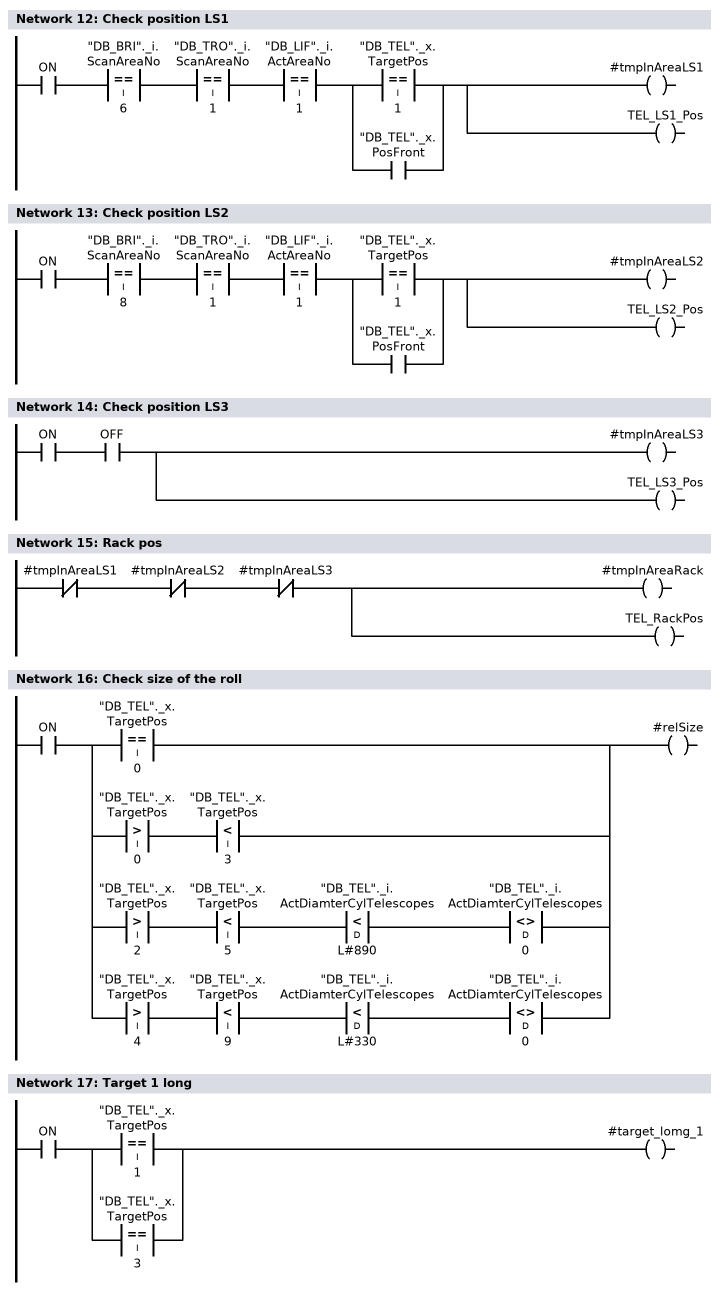
[picture p309: Axis_TEL_Control networks 12-17]
NETWORK
TITLE = Check position LS1
      A     "ON";
      A(;
      L     "DB_BRI"._i.ScanAreaNo;
      L     6;
      ==I;
      );
      A(;
      L     "DB_TRO"._i.ScanAreaNo;
      L     1;
      ==I;
      );
      A(;
      L     "DB_LIF"._i.ActAreaNo;
      L     1;
      ==I;
      );
      A(;
      O(;
      L     "DB_TEL"._x.TargetPos;
      L     1;
      ==I;
      );
      O     "DB_TEL"._x.PosFront;
      );
      =     #tmpInAreaLS1;
      =     "TEL_LS1_Pos";
NETWORK
TITLE = Check position LS2
      A     "ON";
      A(;
      L     "DB_BRI"._i.ScanAreaNo;
      L     8;
      ==I;
      );
      A(;
      L     "DB_TRO"._i.ScanAreaNo;
      L     1;
      ==I;
      );
      A(;
      L     "DB_LIF"._i.ActAreaNo;
      L     1;
      ==I;
      );
      A(;
      O(;
      L     "DB_TEL"._x.TargetPos;
      L     1;
      ==I;
      );
      O     "DB_TEL"._x.PosFront;
      );
      =     #tmpInAreaLS2;
      =     "TEL_LS2_Pos";
NETWORK
TITLE = Check position LS3
      A     "ON";
      A     "OFF";
      =     #tmpInAreaLS3;
      =     "TEL_LS3_Pos";
NETWORK
TITLE = Rack pos
      AN    #tmpInAreaLS1;
      AN    #tmpInAreaLS2;
      AN    #tmpInAreaLS3;
      =     #tmpInAreaRack;
      =     "TEL_RackPos";
NETWORK
TITLE = Check size of the roll
      A     "ON";
      A(;
      O(;
      L     "DB_TEL"._x.TargetPos;
      L     0;
      ==I;
      );
      O;
      A(;
      L     "DB_TEL"._x.TargetPos;
      L     0;
      >I;
      );
      A(;
      L     "DB_TEL"._x.TargetPos;
      L     3;
      <I;
      );
      O;
      A(;
      L     "DB_TEL"._x.TargetPos;
      L     2;
      >I;
      );
      A(;
      L     "DB_TEL"._x.TargetPos;
      L     5;
      <I;
      );
      A(;
      L     "DB_TEL"._i.ActDiamterCylTelescopes;
      L     L#890;
      <D;
      );
      A(;
      L     "DB_TEL"._i.ActDiamterCylTelescopes;
      L     0;
      <>D;
      );
      O;
      A(;
      L     "DB_TEL"._x.TargetPos;
      L     4;
      >I;
      );
      A(;
      L     "DB_TEL"._x.TargetPos;
      L     9;
      <I;
      );
      A(;
      L     "DB_TEL"._i.ActDiamterCylTelescopes;
      L     L#330;
      <D;
      );
      A(;
      L     "DB_TEL"._i.ActDiamterCylTelescopes;
      L     0;
      <>D;
      );
      );
      =     #relSize;
NETWORK
TITLE = Target 1 long
      A     "ON";
      A(;
      O(;
      L     "DB_TEL"._x.TargetPos;
      L     1;
      ==I;
      );
      O(;
      L     "DB_TEL"._x.TargetPos;
      L     3;
      ==I;
      );
      );
      =     #target_lomg_1;
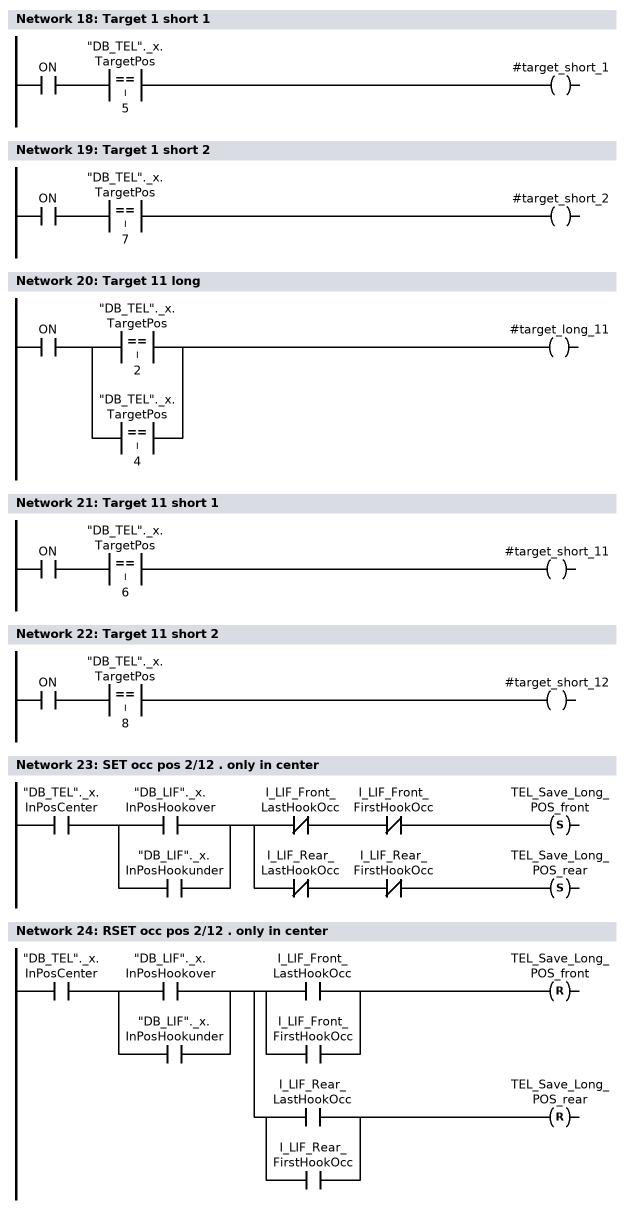
NETWORK
TITLE = Target 1 short 1
      A     "ON";
      A(;
      L     "DB_TEL"._x.TargetPos;
      L     5;
      ==I;
      );
      =     #target_short_1;
NETWORK
TITLE = Target 1 short 2
      A     "ON";
      A(;
      L     "DB_TEL"._x.TargetPos;
      L     7;
      ==I;
      );
      =     #target_short_2;
NETWORK
TITLE = Target 11 long
      A     "ON";
      A(;
      O(;
      L     "DB_TEL"._x.TargetPos;
      L     2;
      ==I;
      );
      O(;
      L     "DB_TEL"._x.TargetPos;
      L     4;
      ==I;
      );
      );
      =     #target_long_11;
NETWORK
TITLE = Target 11 short 1
      A     "ON";
      A(;
      L     "DB_TEL"._x.TargetPos;
      L     6;
      ==I;
      );
      =     #target_short_11;
NETWORK
TITLE = Target 11 short 2
      A     "ON";
      A(;
      L     "DB_TEL"._x.TargetPos;
      L     8;
      ==I;
      );
      =     #target_short_12;
NETWORK
TITLE = SET occ pos 2/12 . only in center
      A     "DB_TEL"._x.InPosCenter;
      A(;
      O     "DB_LIF"._x.InPosHookover;
      O     "DB_LIF"._x.InPosHookunder;
      );
      =     L 20.0;
      A     L 20.0;
      AN    "I_LIF_Front_LastHookOcc";
      AN    "I_LIF_Front_FirstHookOcc";
      S     "TEL_Save_Long_POS_front";
      A     L 20.0;
      AN    "I_LIF_Rear_LastHookOcc";
      AN    "I_LIF_Rear_FirstHookOcc";
      S     "TEL_Save_Long_POS_rear";
NETWORK
TITLE = RSET occ pos 2/12 . only in center
      A     "DB_TEL"._x.InPosCenter;
      A(;
      O     "DB_LIF"._x.InPosHookover;
      O     "DB_LIF"._x.InPosHookunder;
      );
      =     L 20.0;
      A     L 20.0;
      A(;
      O     "I_LIF_Front_LastHookOcc";
      O     "I_LIF_Front_FirstHookOcc";
      );
      R     "TEL_Save_Long_POS_front";
      A     L 20.0;
      A(;
      O     "I_LIF_Rear_LastHookOcc";
      O     "I_LIF_Rear_FirstHookOcc";
      );
      R     "TEL_Save_Long_POS_rear";
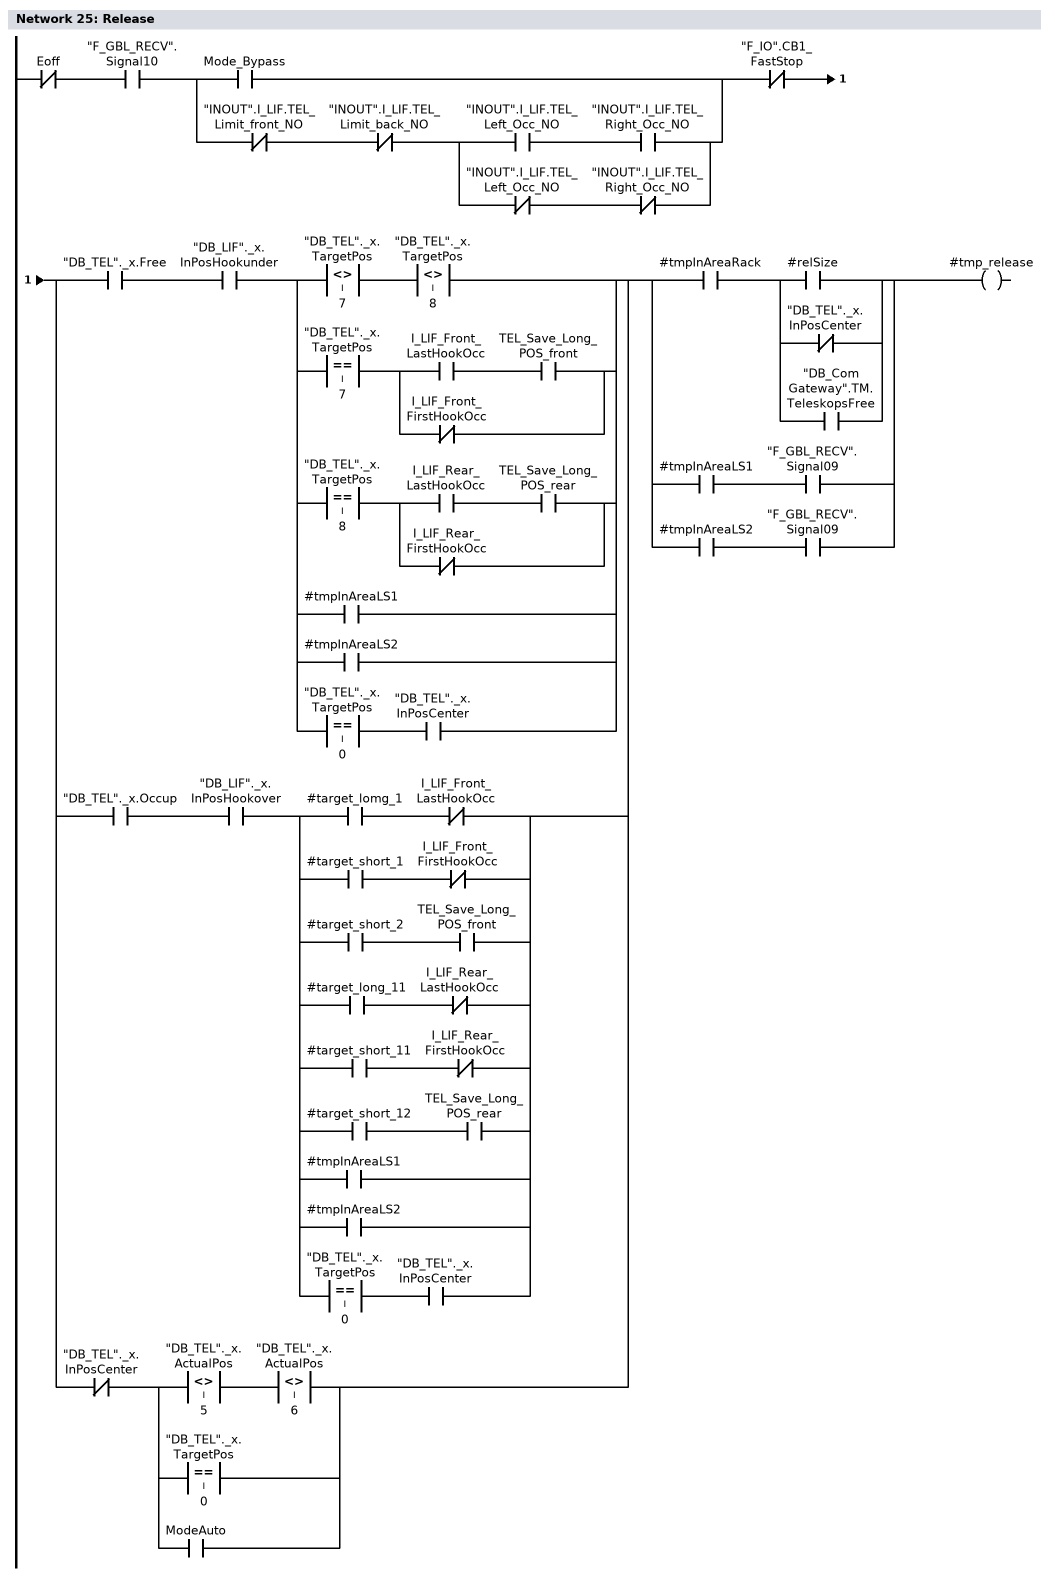
NETWORK
TITLE = Release
//DB400.DBX43.0 LIFT Wago
      AN    "Eoff";
      A     "F_GBL_RECV".Signal10;
      A(;
      O     "Mode_Bypass";
      O;
      AN    "INOUT".I_LIF.TEL_Limit_front_NO;
      AN    "INOUT".I_LIF.TEL_Limit_back_NO;
      A(;
      A     "INOUT".I_LIF.TEL_Left_Occ_NO;
      A     "INOUT".I_LIF.TEL_Right_Occ_NO;
      O;
      AN    "INOUT".I_LIF.TEL_Left_Occ_NO;
      AN    "INOUT".I_LIF.TEL_Right_Occ_NO;
      );
      );
      AN    "F_IO".CB1_FastStop;
      A(;
      A     "DB_TEL"._x.Free;
      A     "DB_LIF"._x.InPosHookunder;
      A(;
      A(;
      L     "DB_TEL"._x.TargetPos;
      L     7;
      <>I;
      );
      A(;
      L     "DB_TEL"._x.TargetPos;
      L     8;
      <>I;
      );
      O;
      A(;
      L     "DB_TEL"._x.TargetPos;
      L     7;
      ==I;
      );
      A(;
      A     "I_LIF_Front_LastHookOcc";
      A     "TEL_Save_Long_POS_front";
      ON    "I_LIF_Front_FirstHookOcc";
      );
      O;
      A(;
      L     "DB_TEL"._x.TargetPos;
      L     8;
      ==I;
      );
      A(;
      A     "I_LIF_Rear_LastHookOcc";
      A     "TEL_Save_Long_POS_rear";
      ON    "I_LIF_Rear_FirstHookOcc";
      );
      O     #tmpInAreaLS1;
      O     #tmpInAreaLS2;
      O;
      A(;
      L     "DB_TEL"._x.TargetPos;
      L     0;
      ==I;
      );
      A     "DB_TEL"._x.InPosCenter;
      );
      O;
      A     "DB_TEL"._x.Occup;
      A     "DB_LIF"._x.InPosHookover;
      A(;
      A     #target_lomg_1;
      AN    "I_LIF_Front_LastHookOcc";
      O;
      A     #target_short_1;
      AN    "I_LIF_Front_FirstHookOcc";
      O;
      A     #target_short_2;
      A     "TEL_Save_Long_POS_front";
      O;
      A     #target_long_11;
      AN    "I_LIF_Rear_LastHookOcc";
      O;
      A     #target_short_11;
      AN    "I_LIF_Rear_FirstHookOcc";
      O;
      A     #target_short_12;
      A     "TEL_Save_Long_POS_rear";
      O     #tmpInAreaLS1;
      O     #tmpInAreaLS2;
      O;
      A(;
      L     "DB_TEL"._x.TargetPos;
      L     0;
      ==I;
      );
      A     "DB_TEL"._x.InPosCenter;
      );
      O;
      AN    "DB_TEL"._x.InPosCenter;
      A(;
      A(;
      L     "DB_TEL"._x.ActualPos;
      L     5;
      <>I;
      );
      A(;
      L     "DB_TEL"._x.ActualPos;
      L     6;
      <>I;
      );
      O(;
      L     "DB_TEL"._x.TargetPos;
      L     0;
      ==I;
      );
      O     "ModeAuto";
      );
      );
      A(;
      A     #tmpInAreaRack;
      A(;
      O     #relSize;
      ON    "DB_TEL"._x.InPosCenter;
      O     "DB_ComGateway".TM.TeleskopsFree;
      );
      O;
      A     #tmpInAreaLS1;
      A     "F_GBL_RECV".Signal09;
      O;
      A     #tmpInAreaLS2;
      A     "F_GBL_RECV".Signal09;
      );
      =     #tmp_release;
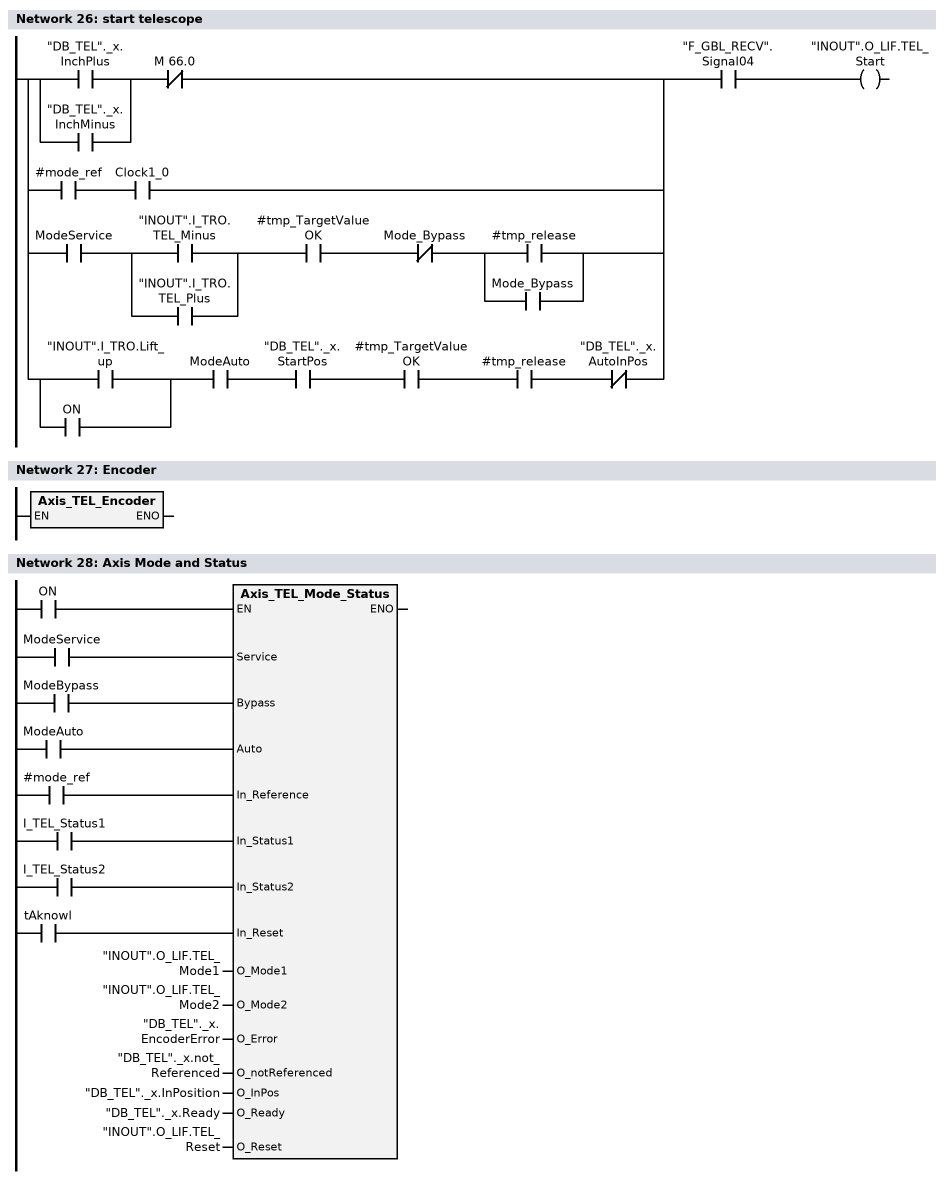
NETWORK
TITLE = start telescope 
      A(;
      A(;
      O     "DB_TEL"._x.InchPlus;
      O     "DB_TEL"._x.InchMinus;
      );
      AN    M 66.0;
      O;
      A     #mode_ref;
      A     "Clock1_0";
      O;
      A     "ModeService";
      A(;
      O     "INOUT".I_TRO.TEL_Minus;
      O     "INOUT".I_TRO.TEL_Plus;
      );
      A     #tmp_TargetValueOK;
      AN    "Mode_Bypass";
      A(;
      O     #tmp_release;
      O     "Mode_Bypass";
      );
      O;
      A(;
      O     "INOUT".I_TRO.Lift_up;
      O     "ON";
      );
      A     "ModeAuto";
      A     "DB_TEL"._x.StartPos;
      A     #tmp_TargetValueOK;
      A     #tmp_release;
      AN    "DB_TEL"._x.AutoInPos;
      );
      A     "F_GBL_RECV".Signal04;
      =     "INOUT".O_LIF.TEL_Start;
NETWORK
TITLE = Encoder
      CALL  "Axis_TEL_Encoder";
      NOP   0;
NETWORK
TITLE = Axis Mode and Status
      A     "ModeService";
      =     L 20.0;
      BLD   103;
      A     "ModeBypass";
      =     L 20.1;
      BLD   103;
      A     "ModeAuto";
      =     L 20.2;
      BLD   103;
      A     #mode_ref;
      =     L 20.3;
      BLD   103;
      A     "I_TEL_Status1";
      =     L 20.4;
      BLD   103;
      A     "I_TEL_Status2";
      =     L 20.5;
      BLD   103;
      A     "tAknowl";
      =     L 20.6;
      BLD   103;
      A     "ON";
      JNB   _00b;
      CALL  "Axis_TEL_Mode_Status" (
           Service                  := L 20.0,
           Bypass                   := L 20.1,
           Auto                     := L 20.2,
           In_Reference             := L 20.3,
           In_Status1               := L 20.4,
           In_Status2               := L 20.5,
           In_Reset                 := L 20.6,
           O_Mode1                  := "INOUT".O_LIF.TEL_Mode1,
           O_Mode2                  := "INOUT".O_LIF.TEL_Mode2,
           O_Error                  := "DB_TEL"._x.EncoderError,
           O_notReferenced          := "DB_TEL"._x.not_Referenced,
           O_InPos                  := "DB_TEL"._x.InPosition,
           O_Ready                  := "DB_TEL"._x.Ready,
           O_Reset                  := "INOUT".O_LIF.TEL_Reset);
_00b: NOP   0;
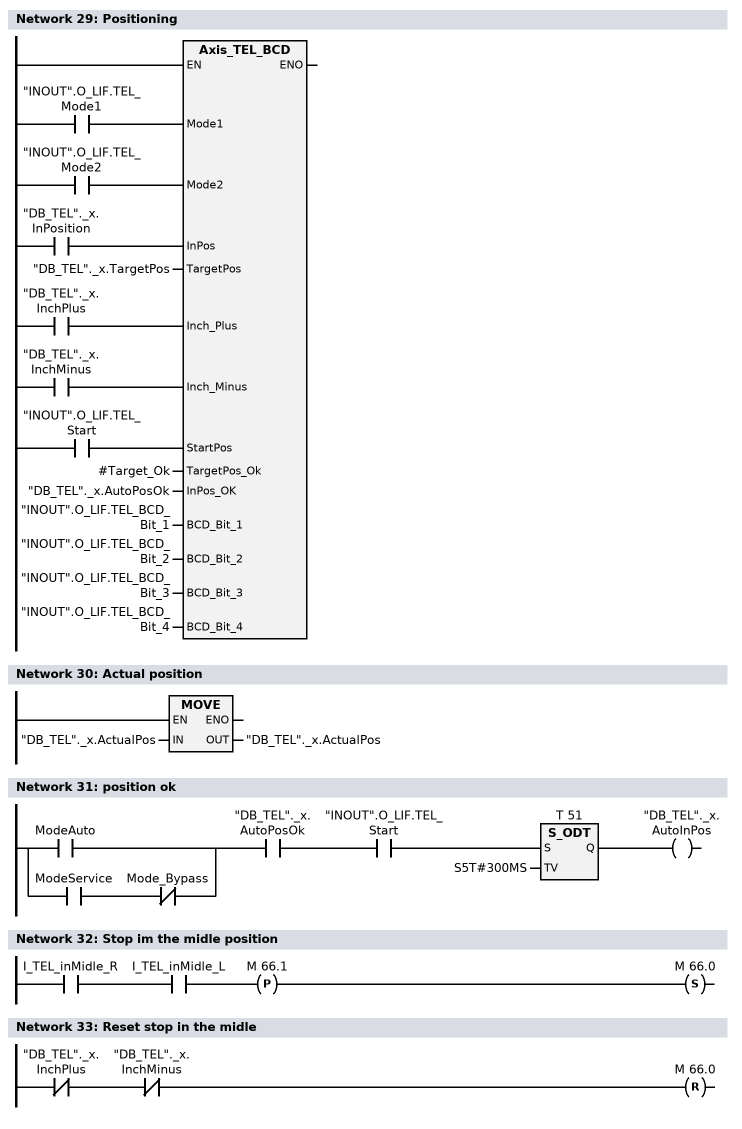
NETWORK
TITLE = Positioning
      A     "INOUT".O_LIF.TEL_Mode1;
      =     L 20.0;
      BLD   103;
      A     "INOUT".O_LIF.TEL_Mode2;
      =     L 20.1;
      BLD   103;
      A     "DB_TEL"._x.InPosition;
      =     L 20.2;
      BLD   103;
      A     "DB_TEL"._x.InchPlus;
      =     L 20.3;
      BLD   103;
      A     "DB_TEL"._x.InchMinus;
      =     L 20.4;
      BLD   103;
      A     "INOUT".O_LIF.TEL_Start;
      =     L 20.5;
      BLD   103;
      CALL  "Axis_TEL_BCD" (
           Mode1                    := L 20.0,
           Mode2                    := L 20.1,
           InPos                    := L 20.2,
           TargetPos                := "DB_TEL"._x.TargetPos,
           Inch_Plus                := L 20.3,
           Inch_Minus               := L 20.4,
           StartPos                 := L 20.5,
           TargetPos_Ok             := #Target_Ok,
           InPos_OK                 := "DB_TEL"._x.AutoPosOk,
           BCD_Bit_1                := "INOUT".O_LIF.TEL_BCD_Bit_1,
           BCD_Bit_2                := "INOUT".O_LIF.TEL_BCD_Bit_2,
           BCD_Bit_3                := "INOUT".O_LIF.TEL_BCD_Bit_3,
           BCD_Bit_4                := "INOUT".O_LIF.TEL_BCD_Bit_4);
      NOP   0;
NETWORK
TITLE = Actual position
      L     "DB_TEL"._x.ActualPos;
      T     "DB_TEL"._x.ActualPos;
      NOP   0;
NETWORK
TITLE = position ok
      A(;
      O     "ModeAuto";
      O;
      A     "ModeService";
      AN    "Mode_Bypass";
      );
      A     "DB_TEL"._x.AutoPosOk;
      A     "INOUT".O_LIF.TEL_Start;
      L     S5T#300MS;
      SD    T 51;
      NOP   0;
      NOP   0;
      NOP   0;
      A     T 51;
      =     "DB_TEL"._x.AutoInPos;
NETWORK
TITLE = Stop im the midle position
      A     "I_TEL_inMidle_R";
      A     "I_TEL_inMidle_L";
      FP    M 66.1;
      S     M 66.0;
NETWORK
TITLE = Reset stop in the midle
      AN    "DB_TEL"._x.InchPlus;
      AN    "DB_TEL"._x.InchMinus;
      R     M 66.0;
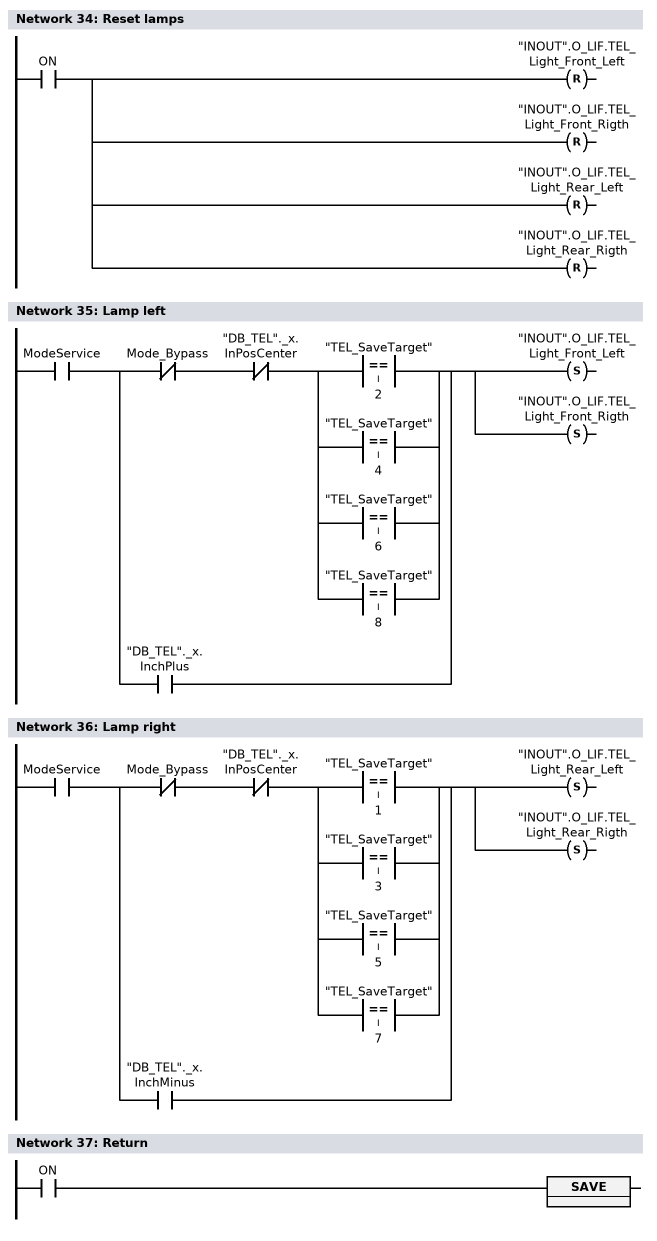
NETWORK
TITLE = Reset lamps
      A     "ON";
      R     "INOUT".O_LIF.TEL_Light_Front_Left;
      R     "INOUT".O_LIF.TEL_Light_Front_Rigth;
      R     "INOUT".O_LIF.TEL_Light_Rear_Left;
      R     "INOUT".O_LIF.TEL_Light_Rear_Rigth;
NETWORK
TITLE = Lamp left
      A     "ModeService";
      A(;
      AN    "Mode_Bypass";
      AN    "DB_TEL"._x.InPosCenter;
      A(;
      O(;
      L     "TEL_SaveTarget";
      L     2;
      ==I;
      );
      O(;
      L     "TEL_SaveTarget";
      L     4;
      ==I;
      );
      O(;
      L     "TEL_SaveTarget";
      L     6;
      ==I;
      );
      O(;
      L     "TEL_SaveTarget";
      L     8;
      ==I;
      );
      );
      O     "DB_TEL"._x.InchPlus;
      );
      S     "INOUT".O_LIF.TEL_Light_Front_Left;
      S     "INOUT".O_LIF.TEL_Light_Front_Rigth;
NETWORK
TITLE = Lamp right
      A     "ModeService";
      A(;
      AN    "Mode_Bypass";
      AN    "DB_TEL"._x.InPosCenter;
      A(;
      O(;
      L     "TEL_SaveTarget";
      L     1;
      ==I;
      );
      O(;
      L     "TEL_SaveTarget";
      L     3;
      ==I;
      );
      O(;
      L     "TEL_SaveTarget";
      L     5;
      ==I;
      );
      O(;
      L     "TEL_SaveTarget";
      L     7;
      ==I;
      );
      );
      O     "DB_TEL"._x.InchMinus;
      );
      S     "INOUT".O_LIF.TEL_Light_Rear_Left;
      S     "INOUT".O_LIF.TEL_Light_Rear_Rigth;
NETWORK
TITLE = Return
      A     "ON";
      SAVE;
END_FUNCTION

FUNCTION "Axis_TEL_Speed" : VOID	// FC 233
VERSION : 0.1
BEGIN
NETWORK
TITLE =
END_FUNCTION

FUNCTION "Axis_TEL_Scan" : VOID	// FC 234
TITLE = Axis TELESCOPES Scan
VERSION : 0.1
VAR_TEMP
  tmp_di_StopWindow : DINT ;
  tmp_di_PosWindow : DINT ;
  tmp_win : DINT ;
  tmp_AreaNo : INT ;
  tmp_InPos : BOOL ;
  tmp_InArea : BOOL ;
  tmp_x_InStopPosMan : BOOL ;
  tmp_x_InStopPosAuto : BOOL ;
  tmp_x_InStopCenterPos : BOOL ;
  tmp_OccFsPos1 : BOOL ;
  tmp_OccBsPos1 : BOOL ;
  tmp_ArriveCenter : BOOL ;
  tmp_MeasureEnd : BOOL ;
  tmp_T56 : BOOL ;
  tmp_T57 : BOOL ;
  tmp_Dir : BOOL ;
END_VAR
BEGIN
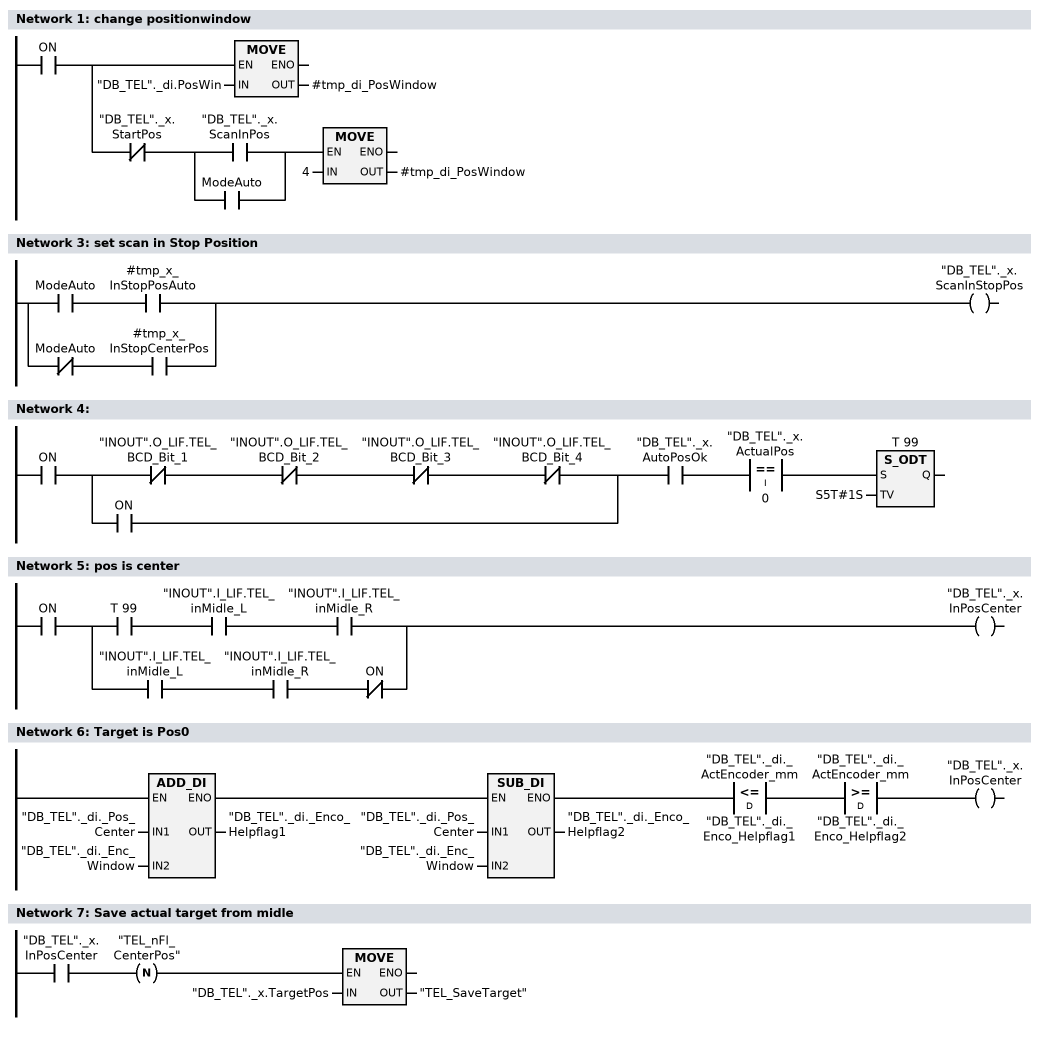
NETWORK
TITLE = change positionwindow
      A     "ON";
      =     L 16.0;
      A     L 16.0;
      JNB   _001;
      L     "DB_TEL"._di.PosWin;
      T     #tmp_di_PosWindow;
_001: NOP   0;
      A     L 16.0;
      AN    "DB_TEL"._x.StartPos;
      A(;
      O     "DB_TEL"._x.ScanInPos;
      O     "ModeAuto";
      );
      JNB   _002;
      L     4;
      T     #tmp_di_PosWindow;
_002: NOP   0;
NETWORK
TITLE = scan telescopes
NETWORK
TITLE = set scan in Stop Position
      A     "ModeAuto";
      A     #tmp_x_InStopPosAuto;
      O;
      AN    "ModeAuto";
      A     #tmp_x_InStopCenterPos;
      =     "DB_TEL"._x.ScanInStopPos;
NETWORK
TITLE =
      A     "ON";
      A(;
      AN    "INOUT".O_LIF.TEL_BCD_Bit_1;
      AN    "INOUT".O_LIF.TEL_BCD_Bit_2;
      AN    "INOUT".O_LIF.TEL_BCD_Bit_3;
      AN    "INOUT".O_LIF.TEL_BCD_Bit_4;
      O     "ON";
      );
      A     "DB_TEL"._x.AutoPosOk;
      A(;
      L     "DB_TEL"._x.ActualPos;
      L     0;
      ==I;
      );
      L     S5T#1S;
      SD    T 99;
      NOP   0;
      NOP   0;
      NOP   0;
      NOP   0;
NETWORK
TITLE = pos is center
//OLD
      A     "ON";
      A(;
      A     T 99;
      A     "INOUT".I_LIF.TEL_inMidle_L;
      A     "INOUT".I_LIF.TEL_inMidle_R;
      O;
      A     "INOUT".I_LIF.TEL_inMidle_L;
      A     "INOUT".I_LIF.TEL_inMidle_R;
      AN    "ON";
      );
      =     "DB_TEL"._x.InPosCenter;
NETWORK
TITLE = Target is Pos0
      A(;
      A(;
      L     "DB_TEL"._di._Pos_Center;
      L     "DB_TEL"._di._Enc_Window;
      +D;
      T     "DB_TEL"._di._Enco_Helpflag1;
      AN    OV;
      SAVE;
      CLR;
      A     BR;
      );
      JNB   _013;
      L     "DB_TEL"._di._Pos_Center;
      L     "DB_TEL"._di._Enc_Window;
      -D;
      T     "DB_TEL"._di._Enco_Helpflag2;
      AN    OV;
      SAVE;
      CLR;
_013: A     BR;
      );
      A(;
      L     "DB_TEL"._di._ActEncoder_mm;
      L     "DB_TEL"._di._Enco_Helpflag1;
      <=D;
      );
      A(;
      L     "DB_TEL"._di._ActEncoder_mm;
      L     "DB_TEL"._di._Enco_Helpflag2;
      >=D;
      );
      =     "DB_TEL"._x.InPosCenter;
NETWORK
TITLE = Save actual target from midle
      A     "DB_TEL"._x.InPosCenter;
      FN    "TEL_nFl_CenterPos";
      JNB   _014;
      L     "DB_TEL"._x.TargetPos;
      T     "TEL_SaveTarget";
_014: NOP   0;
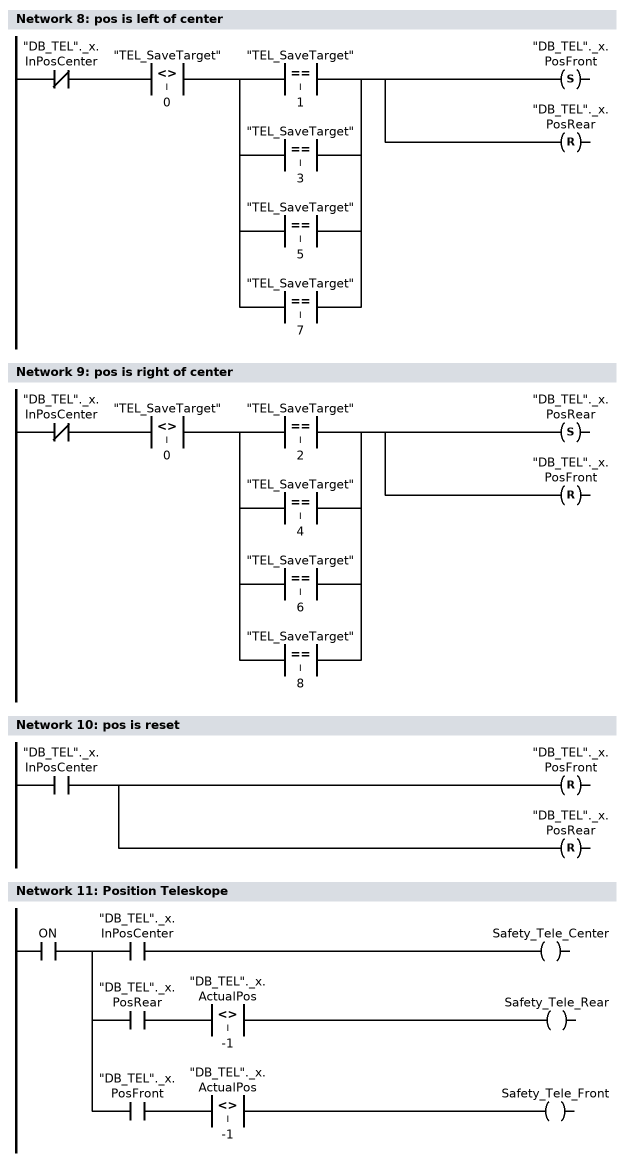
NETWORK
TITLE = pos is left of center
      AN    "DB_TEL"._x.InPosCenter;
      A(;
      L     "TEL_SaveTarget";
      L     0;
      <>I;
      );
      A(;
      O(;
      L     "TEL_SaveTarget";
      L     1;
      ==I;
      );
      O(;
      L     "TEL_SaveTarget";
      L     3;
      ==I;
      );
      O(;
      L     "TEL_SaveTarget";
      L     5;
      ==I;
      );
      O(;
      L     "TEL_SaveTarget";
      L     7;
      ==I;
      );
      );
      S     "DB_TEL"._x.PosFront;
      R     "DB_TEL"._x.PosRear;
NETWORK
TITLE = pos is right of center
      AN    "DB_TEL"._x.InPosCenter;
      A(;
      L     "TEL_SaveTarget";
      L     0;
      <>I;
      );
      A(;
      O(;
      L     "TEL_SaveTarget";
      L     2;
      ==I;
      );
      O(;
      L     "TEL_SaveTarget";
      L     4;
      ==I;
      );
      O(;
      L     "TEL_SaveTarget";
      L     6;
      ==I;
      );
      O(;
      L     "TEL_SaveTarget";
      L     8;
      ==I;
      );
      );
      S     "DB_TEL"._x.PosRear;
      R     "DB_TEL"._x.PosFront;
NETWORK
TITLE = pos is reset
      A     "DB_TEL"._x.InPosCenter;
      R     "DB_TEL"._x.PosFront;
      R     "DB_TEL"._x.PosRear;
NETWORK
TITLE = Position Teleskope
      A     "ON";
      =     L 16.0;
      A     L 16.0;
      A     "DB_TEL"._x.InPosCenter;
      =     "Safety_Tele_Center";
      A     L 16.0;
      A     "DB_TEL"._x.PosRear;
      A(;
      L     "DB_TEL"._x.ActualPos;
      L     -1;
      <>I;
      );
      =     "Safety_Tele_Rear";
      A     L 16.0;
      A     "DB_TEL"._x.PosFront;
      A(;
      L     "DB_TEL"._x.ActualPos;
      L     -1;
      <>I;
      );
      =     "Safety_Tele_Front";
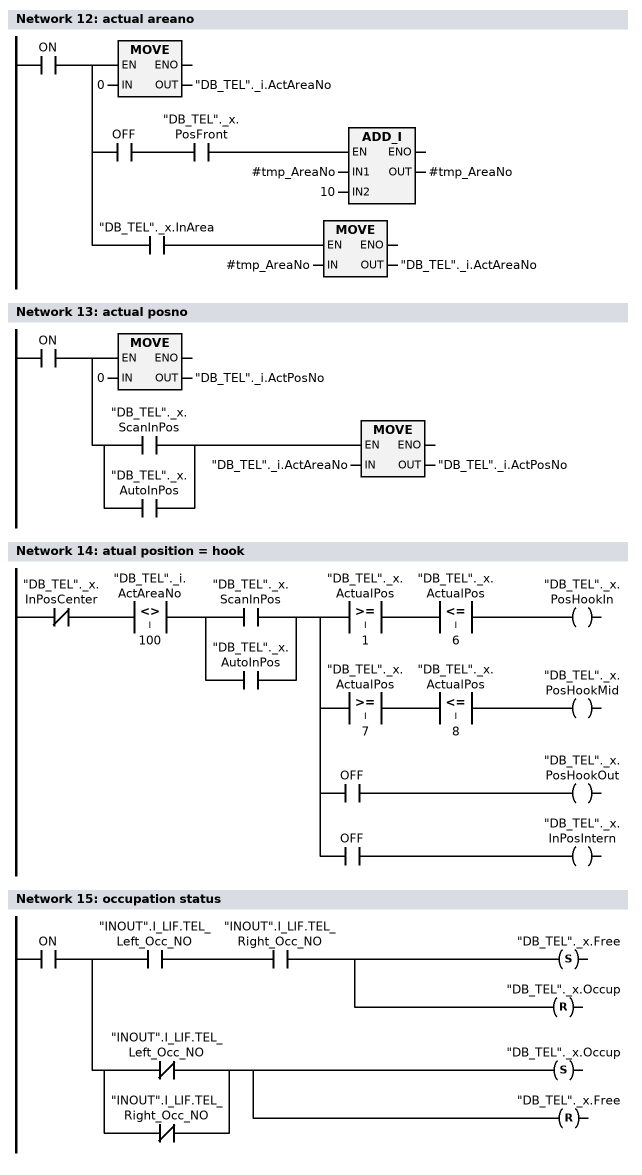
NETWORK
TITLE = actual areano
      A     "ON";
      =     L 16.0;
      A     L 16.0;
      JNB   _015;
      L     0;
      T     "DB_TEL"._i.ActAreaNo;
_015: NOP   0;
      A     L 16.0;
      A     "OFF";
      A     "DB_TEL"._x.PosFront;
      JNB   _016;
      L     #tmp_AreaNo;
      L     10;
      +I;
      T     #tmp_AreaNo;
_016: NOP   0;
      A     L 16.0;
      A     "DB_TEL"._x.InArea;
      JNB   _017;
      L     #tmp_AreaNo;
      T     "DB_TEL"._i.ActAreaNo;
_017: NOP   0;
NETWORK
TITLE = actual posno
      A     "ON";
      =     L 16.0;
      A     L 16.0;
      JNB   _018;
      L     0;
      T     "DB_TEL"._i.ActPosNo;
_018: NOP   0;
      A     L 16.0;
      A(;
      O     "DB_TEL"._x.ScanInPos;
      O     "DB_TEL"._x.AutoInPos;
      );
      JNB   _019;
      L     "DB_TEL"._i.ActAreaNo;
      T     "DB_TEL"._i.ActPosNo;
_019: NOP   0;
NETWORK
TITLE = atual position = hook
      AN    "DB_TEL"._x.InPosCenter;
      A(;
      L     "DB_TEL"._i.ActAreaNo;
      L     100;
      <>I;
      );
      A(;
      O     "DB_TEL"._x.ScanInPos;
      O     "DB_TEL"._x.AutoInPos;
      );
      =     L 16.0;
      A     L 16.0;
      A(;
      L     "DB_TEL"._x.ActualPos;
      L     1;
      >=I;
      );
      A(;
      L     "DB_TEL"._x.ActualPos;
      L     6;
      <=I;
      );
      =     "DB_TEL"._x.PosHookIn;
      A     L 16.0;
      A(;
      L     "DB_TEL"._x.ActualPos;
      L     7;
      >=I;
      );
      A(;
      L     "DB_TEL"._x.ActualPos;
      L     8;
      <=I;
      );
      =     "DB_TEL"._x.PosHookMid;
      A     L 16.0;
      A     "OFF";
      =     "DB_TEL"._x.PosHookOut;
      A     L 16.0;
      A     "OFF";
      =     "DB_TEL"._x.InPosIntern;
NETWORK
TITLE = occupation status
      A     "ON";
      =     L 16.0;
      A     L 16.0;
      A     "INOUT".I_LIF.TEL_Left_Occ_NO;
      A     "INOUT".I_LIF.TEL_Right_Occ_NO;
      S     "DB_TEL"._x.Free;
      R     "DB_TEL"._x.Occup;
      A     L 16.0;
      A(;
      ON    "INOUT".I_LIF.TEL_Left_Occ_NO;
      ON    "INOUT".I_LIF.TEL_Right_Occ_NO;
      );
      S     "DB_TEL"._x.Occup;
      R     "DB_TEL"._x.Free;
NETWORK
TITLE = Check Circumference
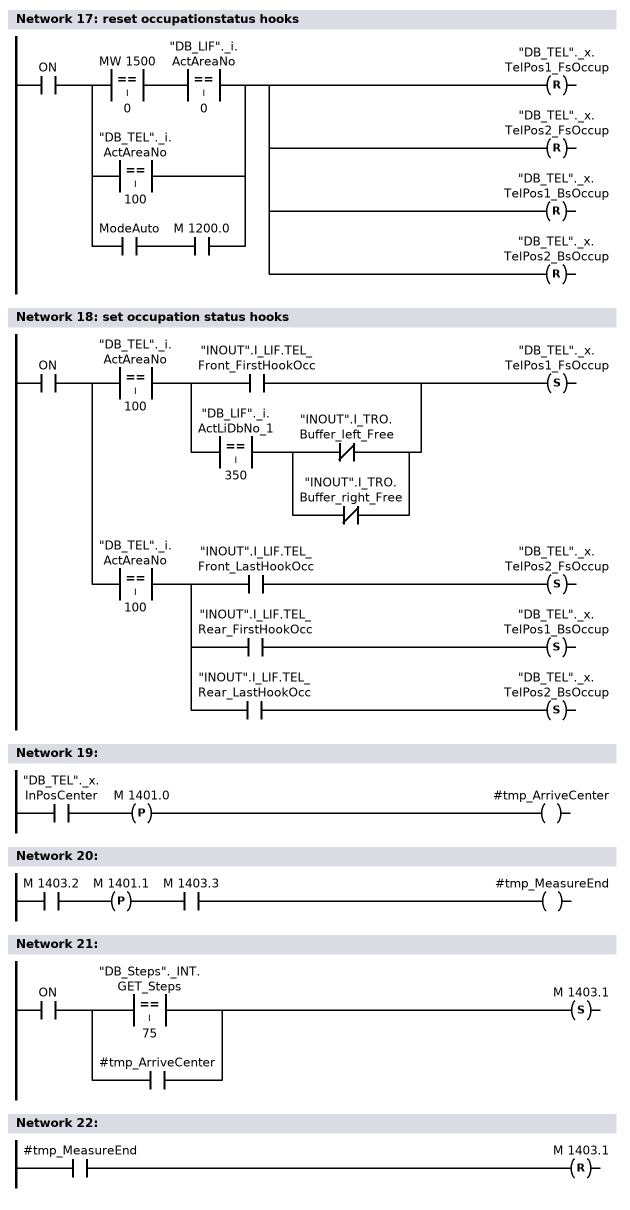
NETWORK
TITLE = reset occupationstatus hooks
      A     "ON";
      A(;
      A(;
      L     MW 1500;
      L     0;
      ==I;
      );
      A(;
      L     "DB_LIF"._i.ActAreaNo;
      L     0;
      ==I;
      );
      O(;
      L     "DB_TEL"._i.ActAreaNo;
      L     100;
      ==I;
      );
      O;
      A     "ModeAuto";
      A     M 1200.0;
      );
      R     "DB_TEL"._x.TelPos1_FsOccup;
      R     "DB_TEL"._x.TelPos2_FsOccup;
      R     "DB_TEL"._x.TelPos1_BsOccup;
      R     "DB_TEL"._x.TelPos2_BsOccup;
NETWORK
TITLE = set occupation status hooks
      A     "ON";
      =     L 16.0;
      A     L 16.0;
      A(;
      L     "DB_TEL"._i.ActAreaNo;
      L     100;
      ==I;
      );
      A(;
      O     "INOUT".I_LIF.TEL_Front_FirstHookOcc;
      O;
      A(;
      L     "DB_LIF"._i.ActLiDbNo_1;
      L     350;
      ==I;
      );
      A(;
      ON    "INOUT".I_TRO.Buffer_left_Free;
      ON    "INOUT".I_TRO.Buffer_right_Free;
      );
      );
      S     "DB_TEL"._x.TelPos1_FsOccup;
      A     L 16.0;
      A(;
      L     "DB_TEL"._i.ActAreaNo;
      L     100;
      ==I;
      );
      =     L 16.1;
      A     L 16.1;
      A     "INOUT".I_LIF.TEL_Front_LastHookOcc;
      S     "DB_TEL"._x.TelPos2_FsOccup;
      A     L 16.1;
      A     "INOUT".I_LIF.TEL_Rear_FirstHookOcc;
      S     "DB_TEL"._x.TelPos1_BsOccup;
      A     L 16.1;
      A     "INOUT".I_LIF.TEL_Rear_LastHookOcc;
      S     "DB_TEL"._x.TelPos2_BsOccup;
NETWORK
TITLE =
      A     "DB_TEL"._x.InPosCenter;
      BLD   100;
      FP    M 1401.0;
      =     #tmp_ArriveCenter;
NETWORK
TITLE =
      A(;
      A     M 1403.2;
      BLD   100;
      FP    M 1401.1;
      );
      A     M 1403.3;
      =     #tmp_MeasureEnd;
NETWORK
TITLE =
      A     "ON";
      A(;
      O(;
      L     "DB_Steps"._INT.GET_Steps;
      L     75;
      ==I;
      );
      O     #tmp_ArriveCenter;
      );
      S     M 1403.1;
NETWORK
TITLE =
      A     #tmp_MeasureEnd;
      R     M 1403.1;
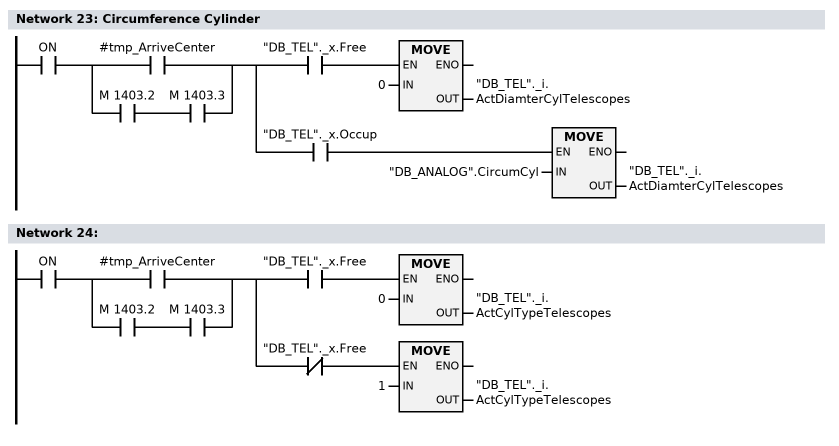
NETWORK
TITLE = Circumference Cylinder
      A     "ON";
      A(;
      O     #tmp_ArriveCenter;
      O;
      A     M 1403.2;
      A     M 1403.3;
      );
      =     L 16.0;
      A     L 16.0;
      A     "DB_TEL"._x.Free;
      JNB   _01a;
      L     0;
      T     "DB_TEL"._i.ActDiamterCylTelescopes;
_01a: NOP   0;
      A     L 16.0;
      A     "DB_TEL"._x.Occup;
      JNB   _01b;
      L     "DB_ANALOG".CircumCyl;
      T     "DB_TEL"._i.ActDiamterCylTelescopes;
_01b: NOP   0;
NETWORK
TITLE =
      A     "ON";
      A(;
      O     #tmp_ArriveCenter;
      O;
      A     M 1403.2;
      A     M 1403.3;
      );
      =     L 16.0;
      A     L 16.0;
      A     "DB_TEL"._x.Free;
      JNB   _01c;
      L     0;
      T     "DB_TEL"._i.ActCylTypeTelescopes;
_01c: NOP   0;
      A     L 16.0;
      AN    "DB_TEL"._x.Free;
      JNB   _01d;
      L     1;
      T     "DB_TEL"._i.ActCylTypeTelescopes;
_01d: NOP   0;
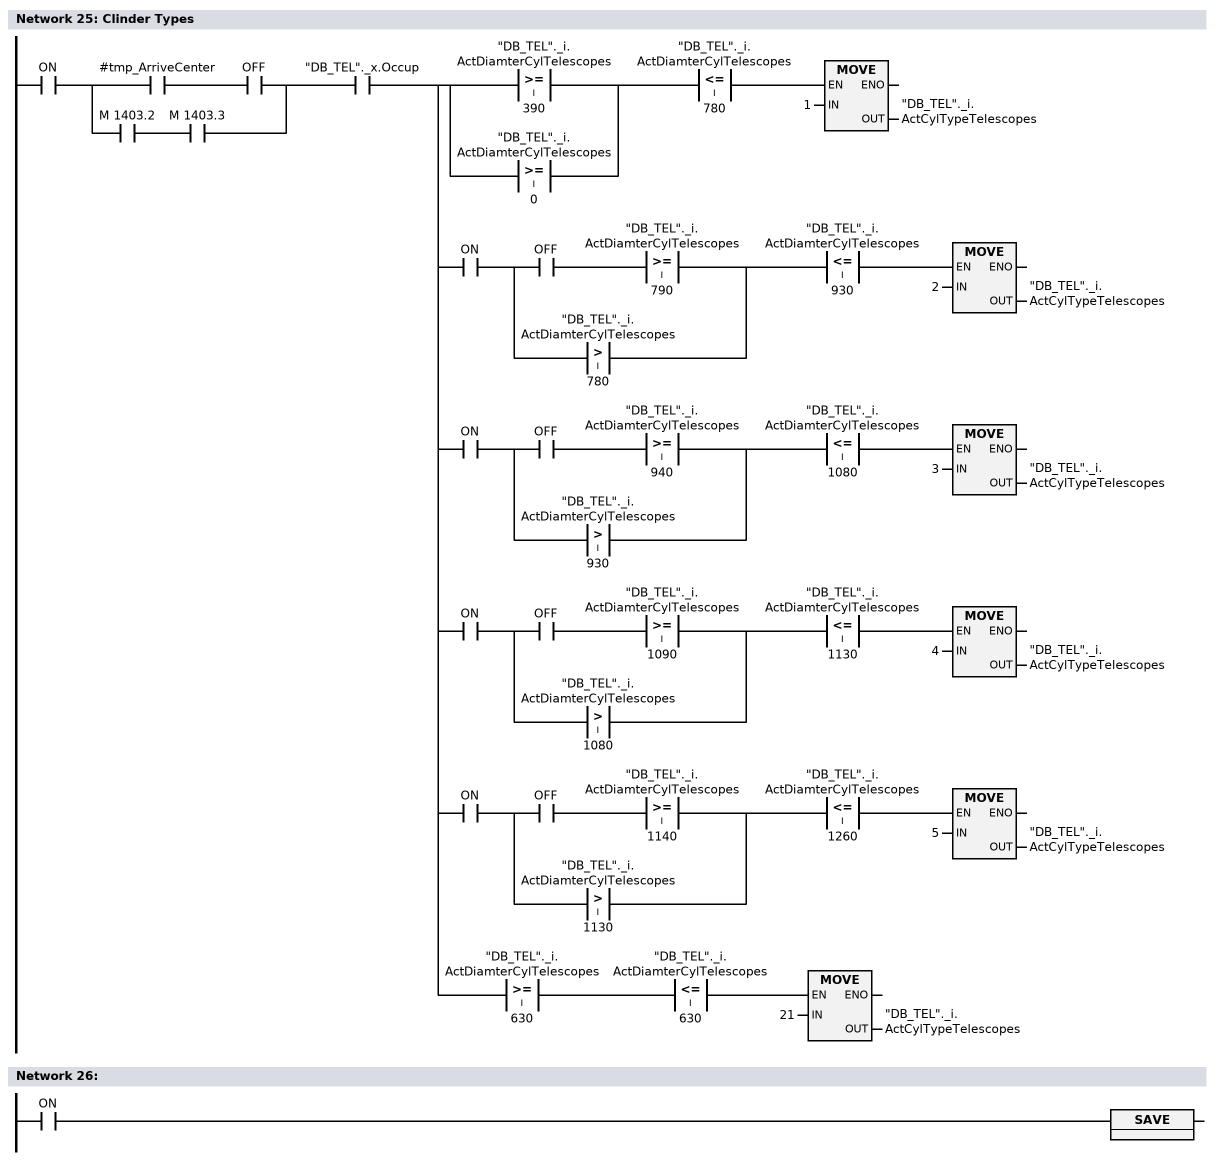
NETWORK
TITLE = Clinder Types
//1 410..760
//2 810..910
//3 960..1060
//4 1110
//5 1160..1260
//21 630 Rasterwalze
      A     "ON";
      A(;
      A     #tmp_ArriveCenter;
      A     "OFF";
      O;
      A     M 1403.2;
      A     M 1403.3;
      );
      A     "DB_TEL"._x.Occup;
      =     L 16.0;
      A     L 16.0;
      A(;
      O(;
      L     "DB_TEL"._i.ActDiamterCylTelescopes;
      L     390;
      >=I;
      );
      O(;
      L     "DB_TEL"._i.ActDiamterCylTelescopes;
      L     0;
      >=I;
      );
      );
      A(;
      L     "DB_TEL"._i.ActDiamterCylTelescopes;
      L     780;
      <=I;
      );
      JNB   _01e;
      L     1;
      T     "DB_TEL"._i.ActCylTypeTelescopes;
_01e: NOP   0;
      A     L 16.0;
      A     "ON";
      A(;
      A     "OFF";
      A(;
      L     "DB_TEL"._i.ActDiamterCylTelescopes;
      L     790;
      >=I;
      );
      O(;
      L     "DB_TEL"._i.ActDiamterCylTelescopes;
      L     780;
      >I;
      );
      );
      A(;
      L     "DB_TEL"._i.ActDiamterCylTelescopes;
      L     930;
      <=I;
      );
      JNB   _01f;
      L     2;
      T     "DB_TEL"._i.ActCylTypeTelescopes;
_01f: NOP   0;
      A     L 16.0;
      A     "ON";
      A(;
      A     "OFF";
      A(;
      L     "DB_TEL"._i.ActDiamterCylTelescopes;
      L     940;
      >=I;
      );
      O(;
      L     "DB_TEL"._i.ActDiamterCylTelescopes;
      L     930;
      >I;
      );
      );
      A(;
      L     "DB_TEL"._i.ActDiamterCylTelescopes;
      L     1080;
      <=I;
      );
      JNB   _020;
      L     3;
      T     "DB_TEL"._i.ActCylTypeTelescopes;
_020: NOP   0;
      A     L 16.0;
      A     "ON";
      A(;
      A     "OFF";
      A(;
      L     "DB_TEL"._i.ActDiamterCylTelescopes;
      L     1090;
      >=I;
      );
      O(;
      L     "DB_TEL"._i.ActDiamterCylTelescopes;
      L     1080;
      >I;
      );
      );
      A(;
      L     "DB_TEL"._i.ActDiamterCylTelescopes;
      L     1130;
      <=I;
      );
      JNB   _021;
      L     4;
      T     "DB_TEL"._i.ActCylTypeTelescopes;
_021: NOP   0;
      A     L 16.0;
      A     "ON";
      A(;
      A     "OFF";
      A(;
      L     "DB_TEL"._i.ActDiamterCylTelescopes;
      L     1140;
      >=I;
      );
      O(;
      L     "DB_TEL"._i.ActDiamterCylTelescopes;
      L     1130;
      >I;
      );
      );
      A(;
      L     "DB_TEL"._i.ActDiamterCylTelescopes;
      L     1260;
      <=I;
      );
      JNB   _022;
      L     5;
      T     "DB_TEL"._i.ActCylTypeTelescopes;
_022: NOP   0;
      A     L 16.0;
      A(;
      L     "DB_TEL"._i.ActDiamterCylTelescopes;
      L     630;
      >=I;
      );
      A(;
      L     "DB_TEL"._i.ActDiamterCylTelescopes;
      L     630;
      <=I;
      );
      JNB   _023;
      L     21;
      T     "DB_TEL"._i.ActCylTypeTelescopes;
_023: NOP   0;
NETWORK
TITLE =
      A     "ON";
      SAVE;
END_FUNCTION

FUNCTION "Axis_TEL_Chk" : VOID	// FC 235
TITLE = Axis TELESCOPE Check
VERSION : 0.1
VAR_TEMP
  tmp_TELTargetFront : BOOL ;
  tmp_TELTargetBack : BOOL ;
END_VAR
BEGIN
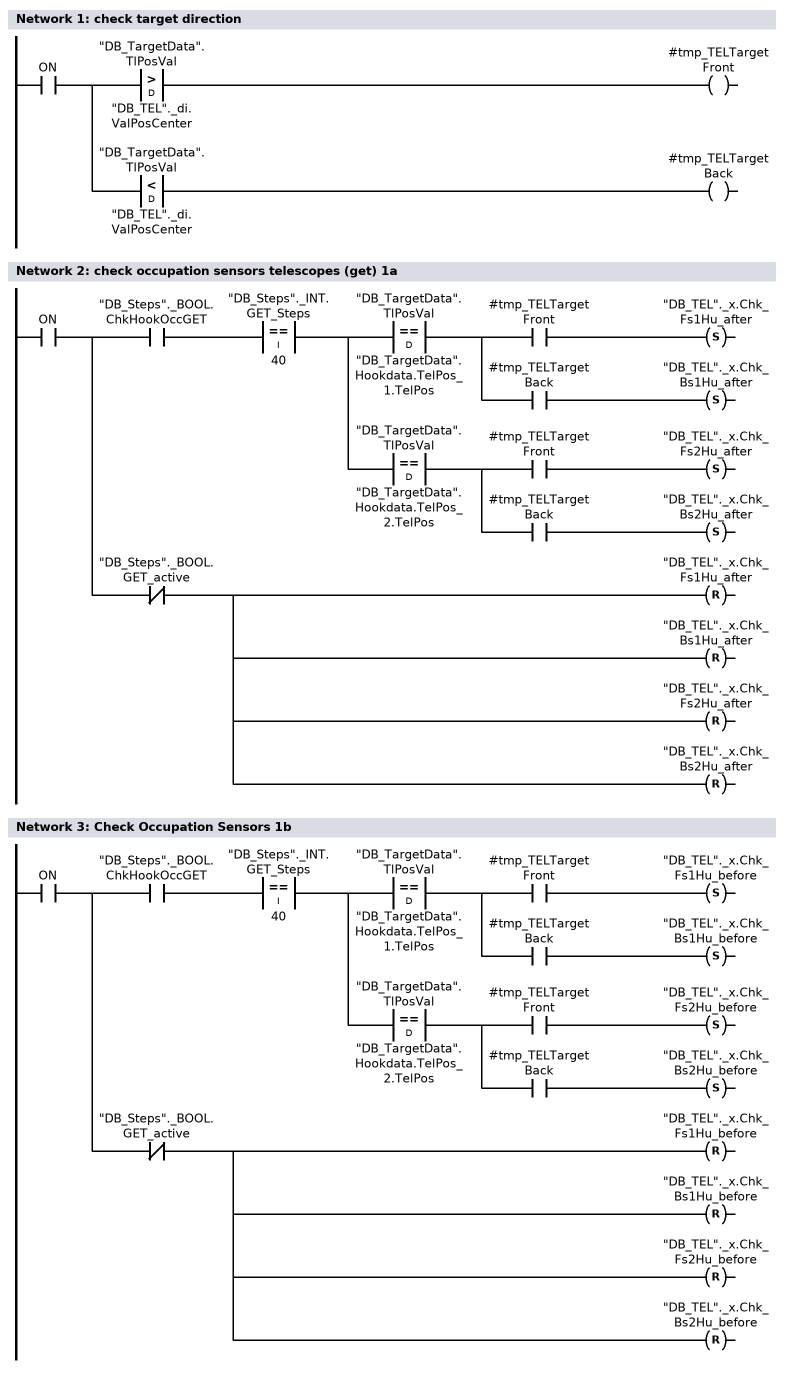
NETWORK
TITLE = check target direction
      A     "ON";
      =     L 1.0;
      A     L 1.0;
      A(;
      L     "DB_TargetData".TlPosVal;
      L     "DB_TEL"._di.ValPosCenter;
      >D;
      );
      =     #tmp_TELTargetFront;
      A     L 1.0;
      A(;
      L     "DB_TargetData".TlPosVal;
      L     "DB_TEL"._di.ValPosCenter;
      <D;
      );
      =     #tmp_TELTargetBack;
NETWORK
TITLE = check occupation sensors telescopes (get) 1a
//GET: Hook under after get
      A     "ON";
      =     L 1.0;
      A     L 1.0;
      A     "DB_Steps"._BOOL.ChkHookOccGET;
      A(;
      L     "DB_Steps"._INT.GET_Steps;
      L     40;
      ==I;
      );
      =     L 1.1;
      A     L 1.1;
      A(;
      L     "DB_TargetData".TlPosVal;
      L     "DB_TargetData".Hookdata.TelPos_1.TelPos;
      ==D;
      );
      =     L 1.2;
      A     L 1.2;
      A     #tmp_TELTargetFront;
      S     "DB_TEL"._x.Chk_Fs1Hu_after;
      A     L 1.2;
      A     #tmp_TELTargetBack;
      S     "DB_TEL"._x.Chk_Bs1Hu_after;
      A     L 1.1;
      A(;
      L     "DB_TargetData".TlPosVal;
      L     "DB_TargetData".Hookdata.TelPos_2.TelPos;
      ==D;
      );
      =     L 1.2;
      A     L 1.2;
      A     #tmp_TELTargetFront;
      S     "DB_TEL"._x.Chk_Fs2Hu_after;
      A     L 1.2;
      A     #tmp_TELTargetBack;
      S     "DB_TEL"._x.Chk_Bs2Hu_after;
      A     L 1.0;
      AN    "DB_Steps"._BOOL.GET_active;
      R     "DB_TEL"._x.Chk_Fs1Hu_after;
      R     "DB_TEL"._x.Chk_Bs1Hu_after;
      R     "DB_TEL"._x.Chk_Fs2Hu_after;
      R     "DB_TEL"._x.Chk_Bs2Hu_after;
NETWORK
TITLE = Check Occupation Sensors 1b
//GET: Hook under before get
      A     "ON";
      =     L 1.0;
      A     L 1.0;
      A     "DB_Steps"._BOOL.ChkHookOccGET;
      A(;
      L     "DB_Steps"._INT.GET_Steps;
      L     40;
      ==I;
      );
      =     L 1.1;
      A     L 1.1;
      A(;
      L     "DB_TargetData".TlPosVal;
      L     "DB_TargetData".Hookdata.TelPos_1.TelPos;
      ==D;
      );
      =     L 1.2;
      A     L 1.2;
      A     #tmp_TELTargetFront;
      S     "DB_TEL"._x.Chk_Fs1Hu_before;
      A     L 1.2;
      A     #tmp_TELTargetBack;
      S     "DB_TEL"._x.Chk_Bs1Hu_before;
      A     L 1.1;
      A(;
      L     "DB_TargetData".TlPosVal;
      L     "DB_TargetData".Hookdata.TelPos_2.TelPos;
      ==D;
      );
      =     L 1.2;
      A     L 1.2;
      A     #tmp_TELTargetFront;
      S     "DB_TEL"._x.Chk_Fs2Hu_before;
      A     L 1.2;
      A     #tmp_TELTargetBack;
      S     "DB_TEL"._x.Chk_Bs2Hu_before;
      A     L 1.0;
      AN    "DB_Steps"._BOOL.GET_active;
      R     "DB_TEL"._x.Chk_Fs1Hu_before;
      R     "DB_TEL"._x.Chk_Bs1Hu_before;
      R     "DB_TEL"._x.Chk_Fs2Hu_before;
      R     "DB_TEL"._x.Chk_Bs2Hu_before;
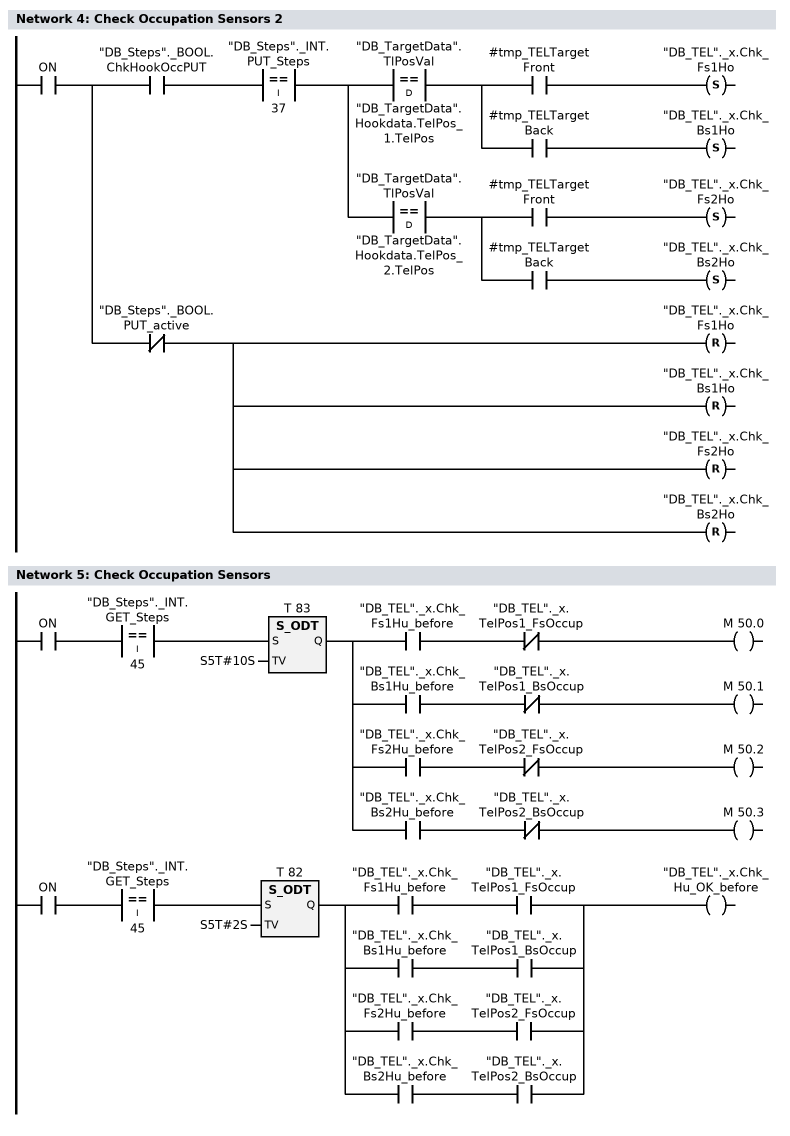
NETWORK
TITLE = Check Occupation Sensors 2
//PUT: Hook over
      A     "ON";
      =     L 1.0;
      A     L 1.0;
      A     "DB_Steps"._BOOL.ChkHookOccPUT;
      A(;
      L     "DB_Steps"._INT.PUT_Steps;
      L     37;
      ==I;
      );
      =     L 1.1;
      A     L 1.1;
      A(;
      L     "DB_TargetData".TlPosVal;
      L     "DB_TargetData".Hookdata.TelPos_1.TelPos;
      ==D;
      );
      =     L 1.2;
      A     L 1.2;
      A     #tmp_TELTargetFront;
      S     "DB_TEL"._x.Chk_Fs1Ho;
      A     L 1.2;
      A     #tmp_TELTargetBack;
      S     "DB_TEL"._x.Chk_Bs1Ho;
      A     L 1.1;
      A(;
      L     "DB_TargetData".TlPosVal;
      L     "DB_TargetData".Hookdata.TelPos_2.TelPos;
      ==D;
      );
      =     L 1.2;
      A     L 1.2;
      A     #tmp_TELTargetFront;
      S     "DB_TEL"._x.Chk_Fs2Ho;
      A     L 1.2;
      A     #tmp_TELTargetBack;
      S     "DB_TEL"._x.Chk_Bs2Ho;
      A     L 1.0;
      AN    "DB_Steps"._BOOL.PUT_active;
      R     "DB_TEL"._x.Chk_Fs1Ho;
      R     "DB_TEL"._x.Chk_Bs1Ho;
      R     "DB_TEL"._x.Chk_Fs2Ho;
      R     "DB_TEL"._x.Chk_Bs2Ho;
NETWORK
TITLE = Check Occupation Sensors
//Check occupation Pos 1 before GET
      A     "ON";
      A(;
      L     "DB_Steps"._INT.GET_Steps;
      L     45;
      ==I;
      );
      =     L 1.0;
      A(;
      A     L 1.0;
      L     S5T#2S;
      SD    T 82;
      NOP   0;
      NOP   0;
      NOP   0;
      A     T 82;
      );
      A(;
      A     "DB_TEL"._x.Chk_Fs1Hu_before;
      A     "DB_TEL"._x.TelPos1_FsOccup;
      O;
      A     "DB_TEL"._x.Chk_Bs1Hu_before;
      A     "DB_TEL"._x.TelPos1_BsOccup;
      O;
      A     "DB_TEL"._x.Chk_Fs2Hu_before;
      A     "DB_TEL"._x.TelPos2_FsOccup;
      O;
      A     "DB_TEL"._x.Chk_Bs2Hu_before;
      A     "DB_TEL"._x.TelPos2_BsOccup;
      );
      =     "DB_TEL"._x.Chk_Hu_OK_before;
      A     L 1.0;
      L     S5T#10S;
      SD    T 83;
      NOP   0;
      NOP   0;
      NOP   0;
      A     T 83;
      =     L 1.1;
      A     L 1.1;
      A     "DB_TEL"._x.Chk_Fs1Hu_before;
      AN    "DB_TEL"._x.TelPos1_FsOccup;
      =     M 50.0;
      A     L 1.1;
      A     "DB_TEL"._x.Chk_Bs1Hu_before;
      AN    "DB_TEL"._x.TelPos1_BsOccup;
      =     M 50.1;
      A     L 1.1;
      A     "DB_TEL"._x.Chk_Fs2Hu_before;
      AN    "DB_TEL"._x.TelPos2_FsOccup;
      =     M 50.2;
      A     L 1.1;
      A     "DB_TEL"._x.Chk_Bs2Hu_before;
      AN    "DB_TEL"._x.TelPos2_BsOccup;
      =     M 50.3;
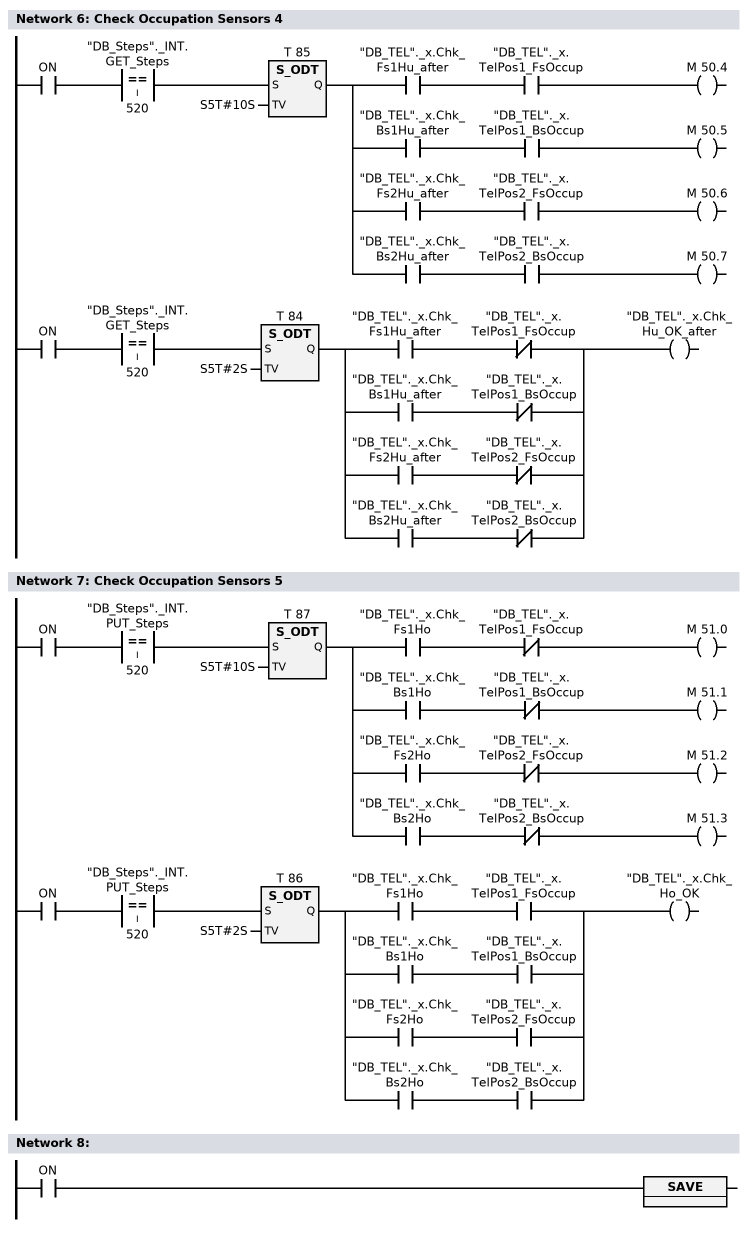
NETWORK
TITLE = Check Occupation Sensors 4
//Check occupation Pos 1 after GET
      A     "ON";
      A(;
      L     "DB_Steps"._INT.GET_Steps;
      L     520;
      ==I;
      );
      =     L 1.0;
      A(;
      A     L 1.0;
      L     S5T#2S;
      SD    T 84;
      NOP   0;
      NOP   0;
      NOP   0;
      A     T 84;
      );
      A(;
      A     "DB_TEL"._x.Chk_Fs1Hu_after;
      AN    "DB_TEL"._x.TelPos1_FsOccup;
      O;
      A     "DB_TEL"._x.Chk_Bs1Hu_after;
      AN    "DB_TEL"._x.TelPos1_BsOccup;
      O;
      A     "DB_TEL"._x.Chk_Fs2Hu_after;
      AN    "DB_TEL"._x.TelPos2_FsOccup;
      O;
      A     "DB_TEL"._x.Chk_Bs2Hu_after;
      AN    "DB_TEL"._x.TelPos2_BsOccup;
      );
      =     "DB_TEL"._x.Chk_Hu_OK_after;
      A     L 1.0;
      L     S5T#10S;
      SD    T 85;
      NOP   0;
      NOP   0;
      NOP   0;
      A     T 85;
      =     L 1.1;
      A     L 1.1;
      A     "DB_TEL"._x.Chk_Fs1Hu_after;
      A     "DB_TEL"._x.TelPos1_FsOccup;
      =     M 50.4;
      A     L 1.1;
      A     "DB_TEL"._x.Chk_Bs1Hu_after;
      A     "DB_TEL"._x.TelPos1_BsOccup;
      =     M 50.5;
      A     L 1.1;
      A     "DB_TEL"._x.Chk_Fs2Hu_after;
      A     "DB_TEL"._x.TelPos2_FsOccup;
      =     M 50.6;
      A     L 1.1;
      A     "DB_TEL"._x.Chk_Bs2Hu_after;
      A     "DB_TEL"._x.TelPos2_BsOccup;
      =     M 50.7;
NETWORK
TITLE = Check Occupation Sensors 5
//Check occupation after PUT
      A     "ON";
      A(;
      L     "DB_Steps"._INT.PUT_Steps;
      L     520;
      ==I;
      );
      =     L 1.0;
      A(;
      A     L 1.0;
      L     S5T#2S;
      SD    T 86;
      NOP   0;
      NOP   0;
      NOP   0;
      A     T 86;
      );
      A(;
      A     "DB_TEL"._x.Chk_Fs1Ho;
      A     "DB_TEL"._x.TelPos1_FsOccup;
      O;
      A     "DB_TEL"._x.Chk_Bs1Ho;
      A     "DB_TEL"._x.TelPos1_BsOccup;
      O;
      A     "DB_TEL"._x.Chk_Fs2Ho;
      A     "DB_TEL"._x.TelPos2_FsOccup;
      O;
      A     "DB_TEL"._x.Chk_Bs2Ho;
      A     "DB_TEL"._x.TelPos2_BsOccup;
      );
      =     "DB_TEL"._x.Chk_Ho_OK;
      A     L 1.0;
      L     S5T#10S;
      SD    T 87;
      NOP   0;
      NOP   0;
      NOP   0;
      A     T 87;
      =     L 1.1;
      A     L 1.1;
      A     "DB_TEL"._x.Chk_Fs1Ho;
      AN    "DB_TEL"._x.TelPos1_FsOccup;
      =     M 51.0;
      A     L 1.1;
      A     "DB_TEL"._x.Chk_Bs1Ho;
      AN    "DB_TEL"._x.TelPos1_BsOccup;
      =     M 51.1;
      A     L 1.1;
      A     "DB_TEL"._x.Chk_Fs2Ho;
      AN    "DB_TEL"._x.TelPos2_FsOccup;
      =     M 51.2;
      A     L 1.1;
      A     "DB_TEL"._x.Chk_Bs2Ho;
      AN    "DB_TEL"._x.TelPos2_BsOccup;
      =     M 51.3;
NETWORK
TITLE =
      A     "ON";
      SAVE;
END_FUNCTION

FUNCTION "Axis_TEL_Mode_Status" : VOID	// FC 237
TITLE = Axis_TEL_Mode_Status
//Mode:
//------------------------------------------------
//Funktion           | DI01 | DI02 | DI03 | DI04 |
//------------------------------------------------
//Keine Betriebsart  |  0   |  0   |  x   |  x   |
//Referenzfahrt      |  1   |  0   |  x   |  x   |
//Handbetrieb        |  0   |  1   |  x   |  x   |
//Positionieren      |  1   |  1   |  x   |  x   |
//Reset              |  x   |  x   |  1   |  0   |
//Start              |  x   |  x   |  0   |  1   |
//
//- 00: No mode // - 01: Tipp mode // - 10: Reference mode // - 11: Auto mode
//
//     
//*******************************************************************************
//    
//Status:
//
//Funktion           |  DO10  | DO11 (GIO12) |
//--------------------------------------------
//Bereit             |    1   |      1       |
//In Position        |    1   |      0       |
//Nicht Referenziert |    0   |      1       |
//Störung            |    0   |      0       |
//
//- 00: Error  // - 01: Not referenced //  - 10: In position  //  - 11: Ready
//
VERSION : 0.1
VAR_INPUT
  Service : BOOL ;
  Bypass : BOOL ;
  Auto : BOOL ;
  In_Reference : BOOL ;
  In_Status1 : BOOL ;
  In_Status2 : BOOL ;
  In_Reset : BOOL ;
END_VAR
VAR_OUTPUT
  O_Mode1 : BOOL ;
  O_Mode2 : BOOL ;
  O_Error : BOOL ;
  O_notReferenced : BOOL ;
  O_InPos : BOOL ;
  O_Ready : BOOL ;
  O_Reset : BOOL ;
END_VAR
VAR_TEMP
  ON : BOOL ;
  OFF : BOOL ;
END_VAR
BEGIN
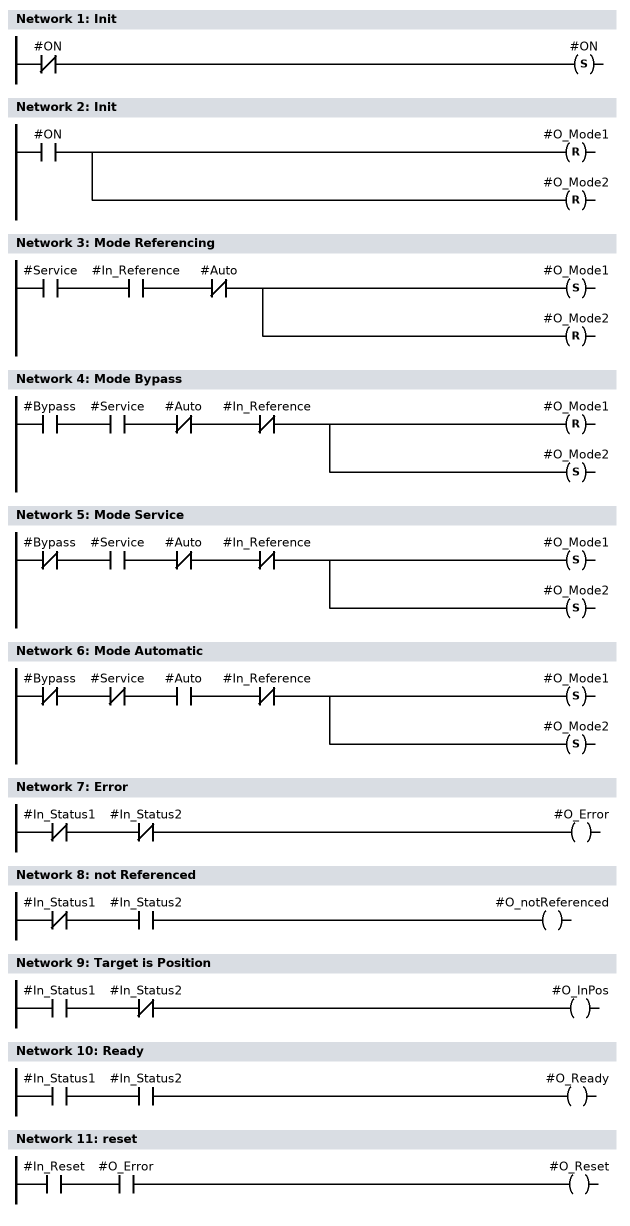
NETWORK
TITLE = Init
      AN    #ON;
      S     #ON;
NETWORK
TITLE = Init
      A     #ON;
      R     #O_Mode1;
      R     #O_Mode2;
NETWORK
TITLE = Mode Referencing
      A     #Service;
      A     #In_Reference;
      AN    #Auto;
      S     #O_Mode1;
      R     #O_Mode2;
NETWORK
TITLE = Mode Bypass
      A     #Bypass;
      A     #Service;
      AN    #Auto;
      AN    #In_Reference;
      R     #O_Mode1;
      S     #O_Mode2;
NETWORK
TITLE = Mode Service
      AN    #Bypass;
      A     #Service;
      AN    #Auto;
      AN    #In_Reference;
      S     #O_Mode1;
      S     #O_Mode2;
NETWORK
TITLE = Mode Automatic
      AN    #Bypass;
      AN    #Service;
      A     #Auto;
      AN    #In_Reference;
      S     #O_Mode1;
      S     #O_Mode2;
NETWORK
TITLE = Error
      AN    #In_Status1;
      AN    #In_Status2;
      =     #O_Error;
NETWORK
TITLE = not Referenced
      AN    #In_Status1;
      A     #In_Status2;
      =     #O_notReferenced;
NETWORK
TITLE = Target is Position
      A     #In_Status1;
      AN    #In_Status2;
      =     #O_InPos;
NETWORK
TITLE = Ready
      A     #In_Status1;
      A     #In_Status2;
      =     #O_Ready;
NETWORK
TITLE = reset
      A     #In_Reset;
      A     #O_Error;
      =     #O_Reset;
END_FUNCTION

FUNCTION "Axis_TEL_BCD" : VOID	// FC 238
//Only in Automatic mode
//
//------------------------------------------------
//Funktion           | DI01 | DI02 | DI03 | DI04 |
//------------------------------------------------
//Keine Betriebsart  |  0   |  0   |  x   |  x   |
//Referenzfahrt      |  1   |  0   |  x   |  x   |
//Handbetrieb        |  0   |  1   |  x   |  x   |
//Positionieren      |  1   |  1   |  x   |  x   |
//Reset              |  x   |  x   |  1   |  0   |
//Start              |  x   |  x   |  0   |  1   |
//
//
//Funktion           | DI10 | DI11 | DI12 | DI13 |
//                   | Bit1 | Bit2 | Bit3 |Bit4
//---------------------------------------------------------------------
//Position0          |  0   |  0   |  0   |  0   |
//Position1          |  1   |  0   |  0   |  0   |
//Position2          |  0   |  1   |  0   |  0   |
//Position3          |  1   |  1   |  0   |  0   |
//Position4          |  0   |  0   |  1   |  0   |
//Position5          |  1   |  0   |  1   |  0   |
//Position6          |  0   |  1   |  1   |  0   |
//Position7          |  1   |  1   |  1   |  0   |
//Position8          |  0   |  0   |  0   |  1   |
//Position9          |  1   |  0   |  0   |  1   |
//
//------------------------------------------------
//
//
VERSION : 0.1
VAR_INPUT
  Mode1 : BOOL ;
  Mode2 : BOOL ;
  InPos : BOOL ;
  TargetPos : INT ;
  Inch_Plus : BOOL ;
  Inch_Minus : BOOL ;
  StartPos : BOOL ;
END_VAR
VAR_OUTPUT
  TargetPos_Ok : BOOL ;
  InPos_OK : BOOL ;
  BCD_Bit_1 : BOOL ;
  BCD_Bit_2 : BOOL ;
  BCD_Bit_3 : BOOL ;
  BCD_Bit_4 : BOOL ;
END_VAR
VAR_TEMP
  ON : BOOL ;
  Auto : BOOL ;
  TargPos : INT ;
  Tipp_Mode : BOOL ;
END_VAR
BEGIN
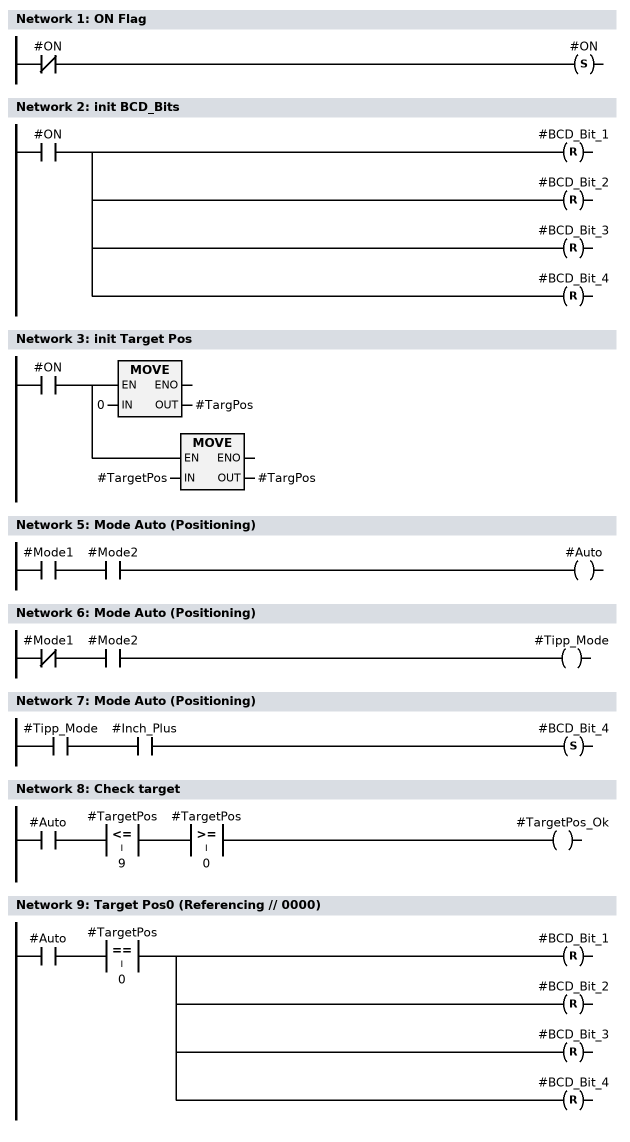
NETWORK
TITLE = ON Flag
      AN    #ON;
      S     #ON;
NETWORK
TITLE = init BCD_Bits
      A     #ON;
      R     #BCD_Bit_1;
      R     #BCD_Bit_2;
      R     #BCD_Bit_3;
      R     #BCD_Bit_4;
NETWORK
TITLE = init Target Pos
      A     #ON;
      =     L 5.0;
      A     L 5.0;
      JNB   _001;
      L     0;
      T     #TargPos;
_001: NOP   0;
      A     L 5.0;
      JNB   _002;
      L     #TargetPos;
      T     #TargPos;
_002: NOP   0;
NETWORK
TITLE = init Actual Pos
NETWORK
TITLE = Mode Auto (Positioning) 
      A     #Mode1;
      A     #Mode2;
      =     #Auto;
NETWORK
TITLE = Mode Auto (Positioning) 
      AN    #Mode1;
      A     #Mode2;
      =     #Tipp_Mode;
NETWORK
TITLE = Mode Auto (Positioning) 
      A     #Tipp_Mode;
      A     #Inch_Plus;
      S     #BCD_Bit_4;
NETWORK
TITLE = Check target
      A     #Auto;
      A(;
      L     #TargetPos;
      L     9;
      <=I;
      );
      A(;
      L     #TargetPos;
      L     0;
      >=I;
      );
      =     #TargetPos_Ok;
NETWORK
TITLE = Target Pos0 (Referencing // 0000)
      A     #Auto;
      A(;
      L     #TargetPos;
      L     0;
      ==I;
      );
      R     #BCD_Bit_1;
      R     #BCD_Bit_2;
      R     #BCD_Bit_3;
      R     #BCD_Bit_4;
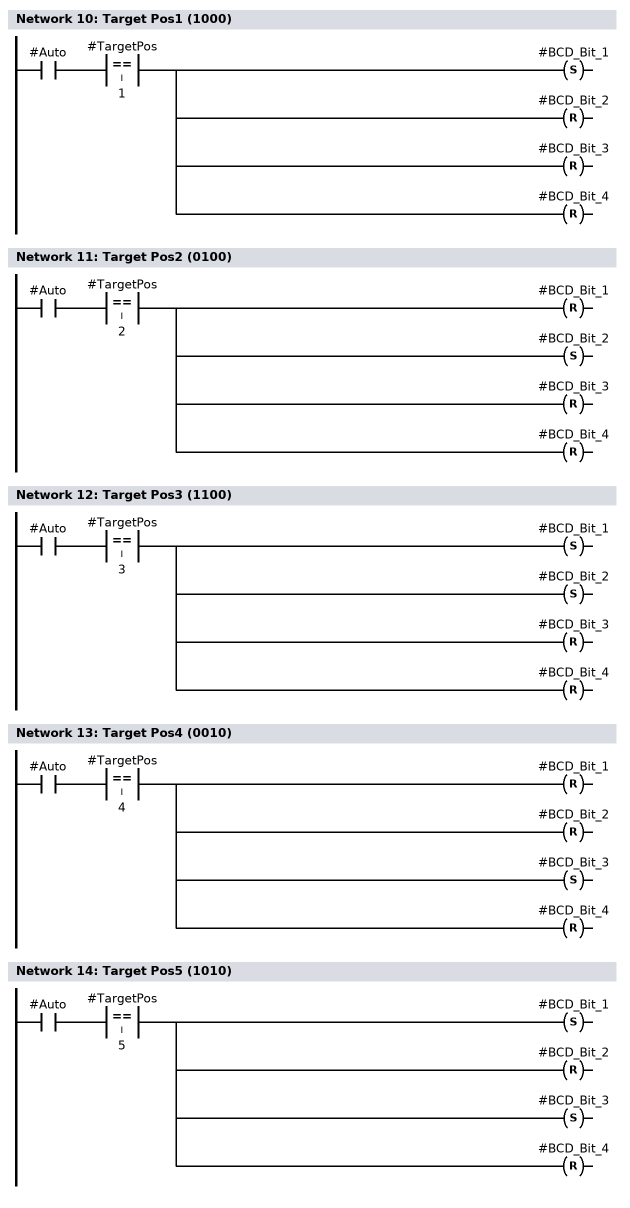
NETWORK
TITLE = Target Pos1 (1000)
      A     #Auto;
      A(;
      L     #TargetPos;
      L     1;
      ==I;
      );
      S     #BCD_Bit_1;
      R     #BCD_Bit_2;
      R     #BCD_Bit_3;
      R     #BCD_Bit_4;
NETWORK
TITLE = Target Pos2 (0100)
      A     #Auto;
      A(;
      L     #TargetPos;
      L     2;
      ==I;
      );
      R     #BCD_Bit_1;
      S     #BCD_Bit_2;
      R     #BCD_Bit_3;
      R     #BCD_Bit_4;
NETWORK
TITLE = Target Pos3 (1100)
      A     #Auto;
      A(;
      L     #TargetPos;
      L     3;
      ==I;
      );
      S     #BCD_Bit_1;
      S     #BCD_Bit_2;
      R     #BCD_Bit_3;
      R     #BCD_Bit_4;
NETWORK
TITLE = Target Pos4 (0010)
      A     #Auto;
      A(;
      L     #TargetPos;
      L     4;
      ==I;
      );
      R     #BCD_Bit_1;
      R     #BCD_Bit_2;
      S     #BCD_Bit_3;
      R     #BCD_Bit_4;
NETWORK
TITLE = Target Pos5 (1010)
      A     #Auto;
      A(;
      L     #TargetPos;
      L     5;
      ==I;
      );
      S     #BCD_Bit_1;
      R     #BCD_Bit_2;
      S     #BCD_Bit_3;
      R     #BCD_Bit_4;
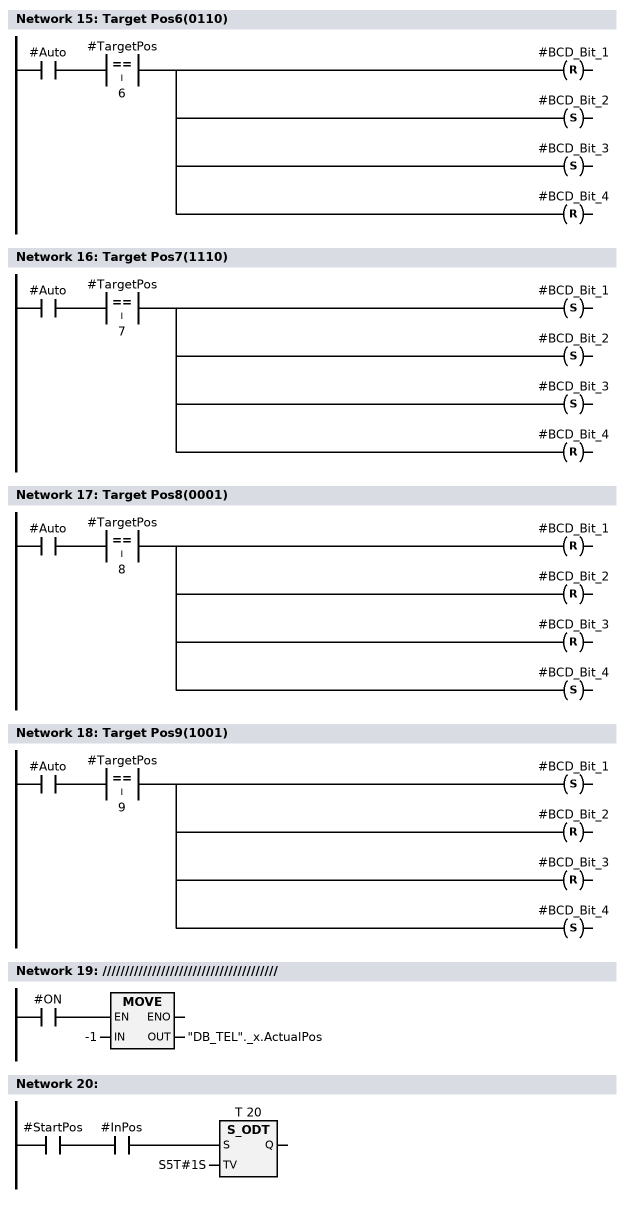
NETWORK
TITLE = Target Pos6(0110)
      A     #Auto;
      A(;
      L     #TargetPos;
      L     6;
      ==I;
      );
      R     #BCD_Bit_1;
      S     #BCD_Bit_2;
      S     #BCD_Bit_3;
      R     #BCD_Bit_4;
NETWORK
TITLE = Target Pos7(1110)
      A     #Auto;
      A(;
      L     #TargetPos;
      L     7;
      ==I;
      );
      S     #BCD_Bit_1;
      S     #BCD_Bit_2;
      S     #BCD_Bit_3;
      R     #BCD_Bit_4;
NETWORK
TITLE = Target Pos8(0001)
      A     #Auto;
      A(;
      L     #TargetPos;
      L     8;
      ==I;
      );
      R     #BCD_Bit_1;
      R     #BCD_Bit_2;
      R     #BCD_Bit_3;
      S     #BCD_Bit_4;
NETWORK
TITLE = Target Pos9(1001)
      A     #Auto;
      A(;
      L     #TargetPos;
      L     9;
      ==I;
      );
      S     #BCD_Bit_1;
      R     #BCD_Bit_2;
      R     #BCD_Bit_3;
      S     #BCD_Bit_4;
NETWORK
TITLE = ///////////////////////////////////////
//no FB ! so set actual pos to -1 if inching or start pos
      A     #ON;
      JNB   _003;
      L     -1;
      T     "DB_TEL"._x.ActualPos;
_003: NOP   0;
NETWORK
TITLE =
      A     #StartPos;
      A     #InPos;
      L     S5T#1S;
      SD    T 20;
      NOP   0;
      NOP   0;
      NOP   0;
      NOP   0;
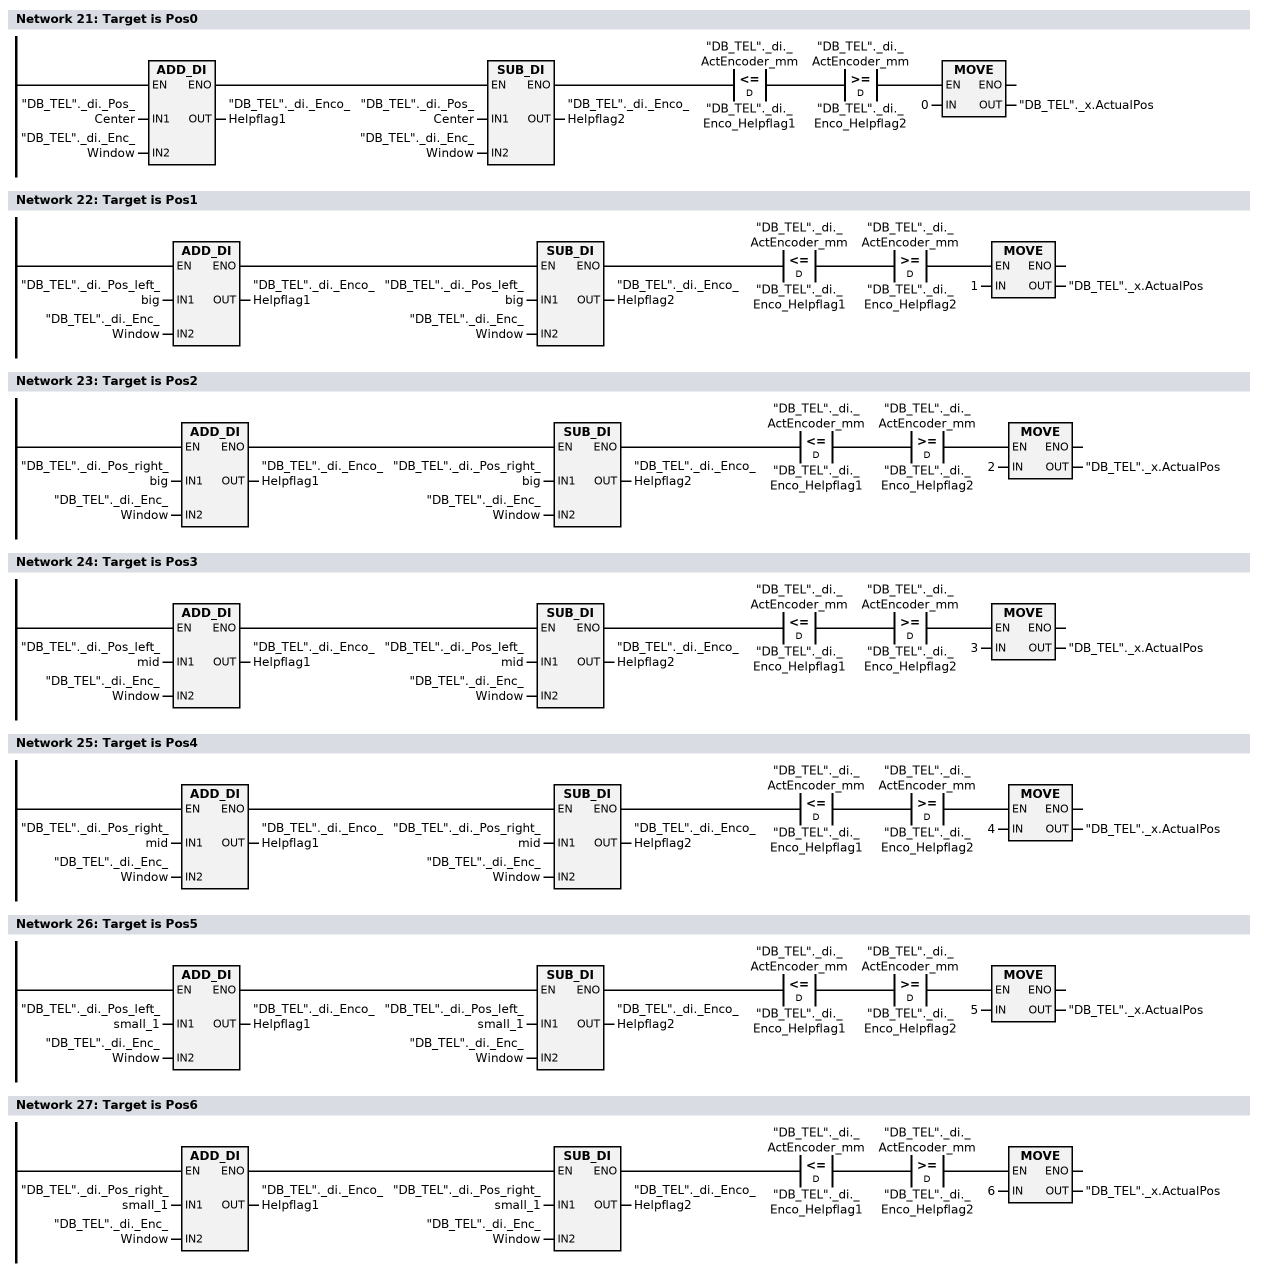
NETWORK
TITLE = Target is Pos0
      A(;
      A(;
      L     "DB_TEL"._di._Pos_Center;
      L     "DB_TEL"._di._Enc_Window;
      +D;
      T     "DB_TEL"._di._Enco_Helpflag1;
      AN    OV;
      SAVE;
      CLR;
      A     BR;
      );
      JNB   _004;
      L     "DB_TEL"._di._Pos_Center;
      L     "DB_TEL"._di._Enc_Window;
      -D;
      T     "DB_TEL"._di._Enco_Helpflag2;
      AN    OV;
      SAVE;
      CLR;
_004: A     BR;
      );
      A(;
      L     "DB_TEL"._di._ActEncoder_mm;
      L     "DB_TEL"._di._Enco_Helpflag1;
      <=D;
      );
      A(;
      L     "DB_TEL"._di._ActEncoder_mm;
      L     "DB_TEL"._di._Enco_Helpflag2;
      >=D;
      );
      JNB   _005;
      L     0;
      T     "DB_TEL"._x.ActualPos;
_005: NOP   0;
NETWORK
TITLE = Target is Pos1
      A(;
      A(;
      L     "DB_TEL"._di._Pos_left_big;
      L     "DB_TEL"._di._Enc_Window;
      +D;
      T     "DB_TEL"._di._Enco_Helpflag1;
      AN    OV;
      SAVE;
      CLR;
      A     BR;
      );
      JNB   _006;
      L     "DB_TEL"._di._Pos_left_big;
      L     "DB_TEL"._di._Enc_Window;
      -D;
      T     "DB_TEL"._di._Enco_Helpflag2;
      AN    OV;
      SAVE;
      CLR;
_006: A     BR;
      );
      A(;
      L     "DB_TEL"._di._ActEncoder_mm;
      L     "DB_TEL"._di._Enco_Helpflag1;
      <=D;
      );
      A(;
      L     "DB_TEL"._di._ActEncoder_mm;
      L     "DB_TEL"._di._Enco_Helpflag2;
      >=D;
      );
      JNB   _007;
      L     1;
      T     "DB_TEL"._x.ActualPos;
_007: NOP   0;
NETWORK
TITLE = Target is Pos2
      A(;
      A(;
      L     "DB_TEL"._di._Pos_right_big;
      L     "DB_TEL"._di._Enc_Window;
      +D;
      T     "DB_TEL"._di._Enco_Helpflag1;
      AN    OV;
      SAVE;
      CLR;
      A     BR;
      );
      JNB   _008;
      L     "DB_TEL"._di._Pos_right_big;
      L     "DB_TEL"._di._Enc_Window;
      -D;
      T     "DB_TEL"._di._Enco_Helpflag2;
      AN    OV;
      SAVE;
      CLR;
_008: A     BR;
      );
      A(;
      L     "DB_TEL"._di._ActEncoder_mm;
      L     "DB_TEL"._di._Enco_Helpflag1;
      <=D;
      );
      A(;
      L     "DB_TEL"._di._ActEncoder_mm;
      L     "DB_TEL"._di._Enco_Helpflag2;
      >=D;
      );
      JNB   _009;
      L     2;
      T     "DB_TEL"._x.ActualPos;
_009: NOP   0;
NETWORK
TITLE = Target is Pos3
      A(;
      A(;
      L     "DB_TEL"._di._Pos_left_mid;
      L     "DB_TEL"._di._Enc_Window;
      +D;
      T     "DB_TEL"._di._Enco_Helpflag1;
      AN    OV;
      SAVE;
      CLR;
      A     BR;
      );
      JNB   _00a;
      L     "DB_TEL"._di._Pos_left_mid;
      L     "DB_TEL"._di._Enc_Window;
      -D;
      T     "DB_TEL"._di._Enco_Helpflag2;
      AN    OV;
      SAVE;
      CLR;
_00a: A     BR;
      );
      A(;
      L     "DB_TEL"._di._ActEncoder_mm;
      L     "DB_TEL"._di._Enco_Helpflag1;
      <=D;
      );
      A(;
      L     "DB_TEL"._di._ActEncoder_mm;
      L     "DB_TEL"._di._Enco_Helpflag2;
      >=D;
      );
      JNB   _00b;
      L     3;
      T     "DB_TEL"._x.ActualPos;
_00b: NOP   0;
NETWORK
TITLE = Target is Pos4
      A(;
      A(;
      L     "DB_TEL"._di._Pos_right_mid;
      L     "DB_TEL"._di._Enc_Window;
      +D;
      T     "DB_TEL"._di._Enco_Helpflag1;
      AN    OV;
      SAVE;
      CLR;
      A     BR;
      );
      JNB   _00c;
      L     "DB_TEL"._di._Pos_right_mid;
      L     "DB_TEL"._di._Enc_Window;
      -D;
      T     "DB_TEL"._di._Enco_Helpflag2;
      AN    OV;
      SAVE;
      CLR;
_00c: A     BR;
      );
      A(;
      L     "DB_TEL"._di._ActEncoder_mm;
      L     "DB_TEL"._di._Enco_Helpflag1;
      <=D;
      );
      A(;
      L     "DB_TEL"._di._ActEncoder_mm;
      L     "DB_TEL"._di._Enco_Helpflag2;
      >=D;
      );
      JNB   _00d;
      L     4;
      T     "DB_TEL"._x.ActualPos;
_00d: NOP   0;
NETWORK
TITLE = Target is Pos5
      A(;
      A(;
      L     "DB_TEL"._di._Pos_left_small_1;
      L     "DB_TEL"._di._Enc_Window;
      +D;
      T     "DB_TEL"._di._Enco_Helpflag1;
      AN    OV;
      SAVE;
      CLR;
      A     BR;
      );
      JNB   _00e;
      L     "DB_TEL"._di._Pos_left_small_1;
      L     "DB_TEL"._di._Enc_Window;
      -D;
      T     "DB_TEL"._di._Enco_Helpflag2;
      AN    OV;
      SAVE;
      CLR;
_00e: A     BR;
      );
      A(;
      L     "DB_TEL"._di._ActEncoder_mm;
      L     "DB_TEL"._di._Enco_Helpflag1;
      <=D;
      );
      A(;
      L     "DB_TEL"._di._ActEncoder_mm;
      L     "DB_TEL"._di._Enco_Helpflag2;
      >=D;
      );
      JNB   _00f;
      L     5;
      T     "DB_TEL"._x.ActualPos;
_00f: NOP   0;
NETWORK
TITLE = Target is Pos6
      A(;
      A(;
      L     "DB_TEL"._di._Pos_right_small_1;
      L     "DB_TEL"._di._Enc_Window;
      +D;
      T     "DB_TEL"._di._Enco_Helpflag1;
      AN    OV;
      SAVE;
      CLR;
      A     BR;
      );
      JNB   _010;
      L     "DB_TEL"._di._Pos_right_small_1;
      L     "DB_TEL"._di._Enc_Window;
      -D;
      T     "DB_TEL"._di._Enco_Helpflag2;
      AN    OV;
      SAVE;
      CLR;
_010: A     BR;
      );
      A(;
      L     "DB_TEL"._di._ActEncoder_mm;
      L     "DB_TEL"._di._Enco_Helpflag1;
      <=D;
      );
      A(;
      L     "DB_TEL"._di._ActEncoder_mm;
      L     "DB_TEL"._di._Enco_Helpflag2;
      >=D;
      );
      JNB   _011;
      L     6;
      T     "DB_TEL"._x.ActualPos;
_011: NOP   0;
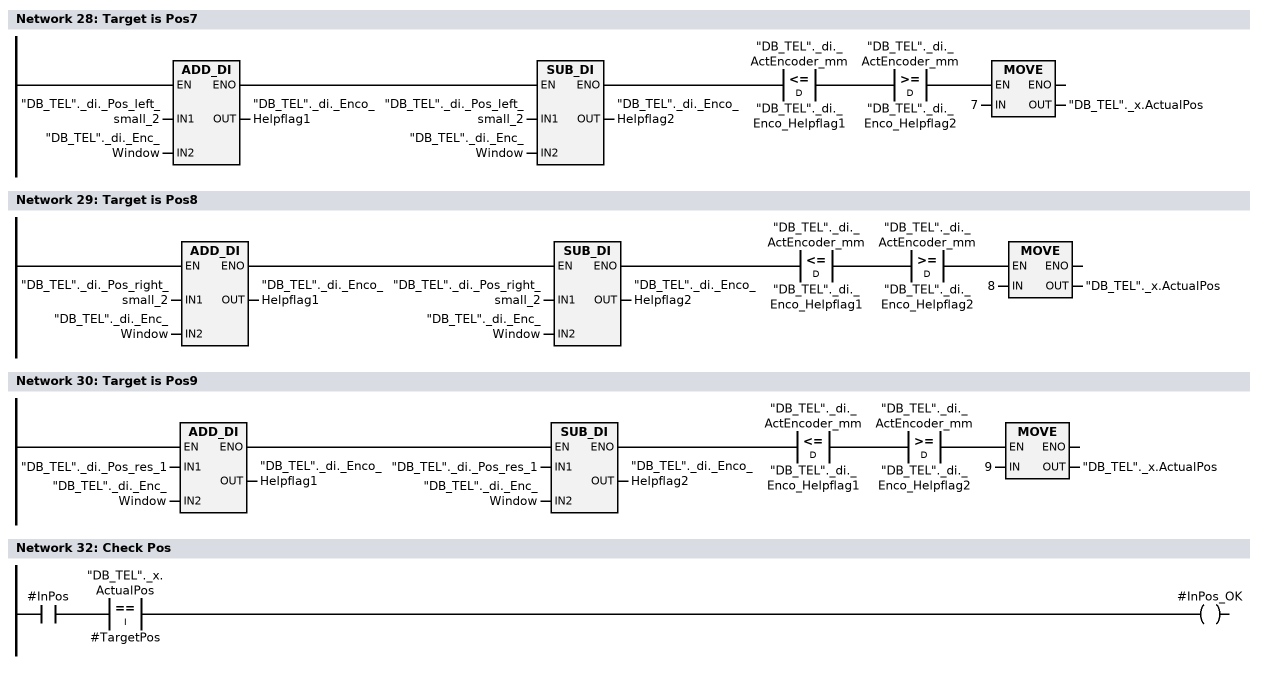
NETWORK
TITLE = Target is Pos7
      A(;
      A(;
      L     "DB_TEL"._di._Pos_left_small_2;
      L     "DB_TEL"._di._Enc_Window;
      +D;
      T     "DB_TEL"._di._Enco_Helpflag1;
      AN    OV;
      SAVE;
      CLR;
      A     BR;
      );
      JNB   _012;
      L     "DB_TEL"._di._Pos_left_small_2;
      L     "DB_TEL"._di._Enc_Window;
      -D;
      T     "DB_TEL"._di._Enco_Helpflag2;
      AN    OV;
      SAVE;
      CLR;
_012: A     BR;
      );
      A(;
      L     "DB_TEL"._di._ActEncoder_mm;
      L     "DB_TEL"._di._Enco_Helpflag1;
      <=D;
      );
      A(;
      L     "DB_TEL"._di._ActEncoder_mm;
      L     "DB_TEL"._di._Enco_Helpflag2;
      >=D;
      );
      JNB   _013;
      L     7;
      T     "DB_TEL"._x.ActualPos;
_013: NOP   0;
NETWORK
TITLE = Target is Pos8
      A(;
      A(;
      L     "DB_TEL"._di._Pos_right_small_2;
      L     "DB_TEL"._di._Enc_Window;
      +D;
      T     "DB_TEL"._di._Enco_Helpflag1;
      AN    OV;
      SAVE;
      CLR;
      A     BR;
      );
      JNB   _014;
      L     "DB_TEL"._di._Pos_right_small_2;
      L     "DB_TEL"._di._Enc_Window;
      -D;
      T     "DB_TEL"._di._Enco_Helpflag2;
      AN    OV;
      SAVE;
      CLR;
_014: A     BR;
      );
      A(;
      L     "DB_TEL"._di._ActEncoder_mm;
      L     "DB_TEL"._di._Enco_Helpflag1;
      <=D;
      );
      A(;
      L     "DB_TEL"._di._ActEncoder_mm;
      L     "DB_TEL"._di._Enco_Helpflag2;
      >=D;
      );
      JNB   _015;
      L     8;
      T     "DB_TEL"._x.ActualPos;
_015: NOP   0;
NETWORK
TITLE = Target is Pos9
      A(;
      A(;
      L     "DB_TEL"._di._Pos_res_1;
      L     "DB_TEL"._di._Enc_Window;
      +D;
      T     "DB_TEL"._di._Enco_Helpflag1;
      AN    OV;
      SAVE;
      CLR;
      A     BR;
      );
      JNB   _016;
      L     "DB_TEL"._di._Pos_res_1;
      L     "DB_TEL"._di._Enc_Window;
      -D;
      T     "DB_TEL"._di._Enco_Helpflag2;
      AN    OV;
      SAVE;
      CLR;
_016: A     BR;
      );
      A(;
      L     "DB_TEL"._di._ActEncoder_mm;
      L     "DB_TEL"._di._Enco_Helpflag1;
      <=D;
      );
      A(;
      L     "DB_TEL"._di._ActEncoder_mm;
      L     "DB_TEL"._di._Enco_Helpflag2;
      >=D;
      );
      JNB   _017;
      L     9;
      T     "DB_TEL"._x.ActualPos;
_017: NOP   0;
NETWORK
TITLE = //////////////////////////////////
NETWORK
TITLE = Check Pos
      A     #InPos;
      A(;
      L     "DB_TEL"._x.ActualPos;
      L     #TargetPos;
      ==I;
      );
      =     #InPos_OK;
END_FUNCTION

FUNCTION "Axis_TEL_Flt_097-112" : VOID	// FC 239
TITLE = Error Telescope 97-112
VERSION : 0.1
BEGIN
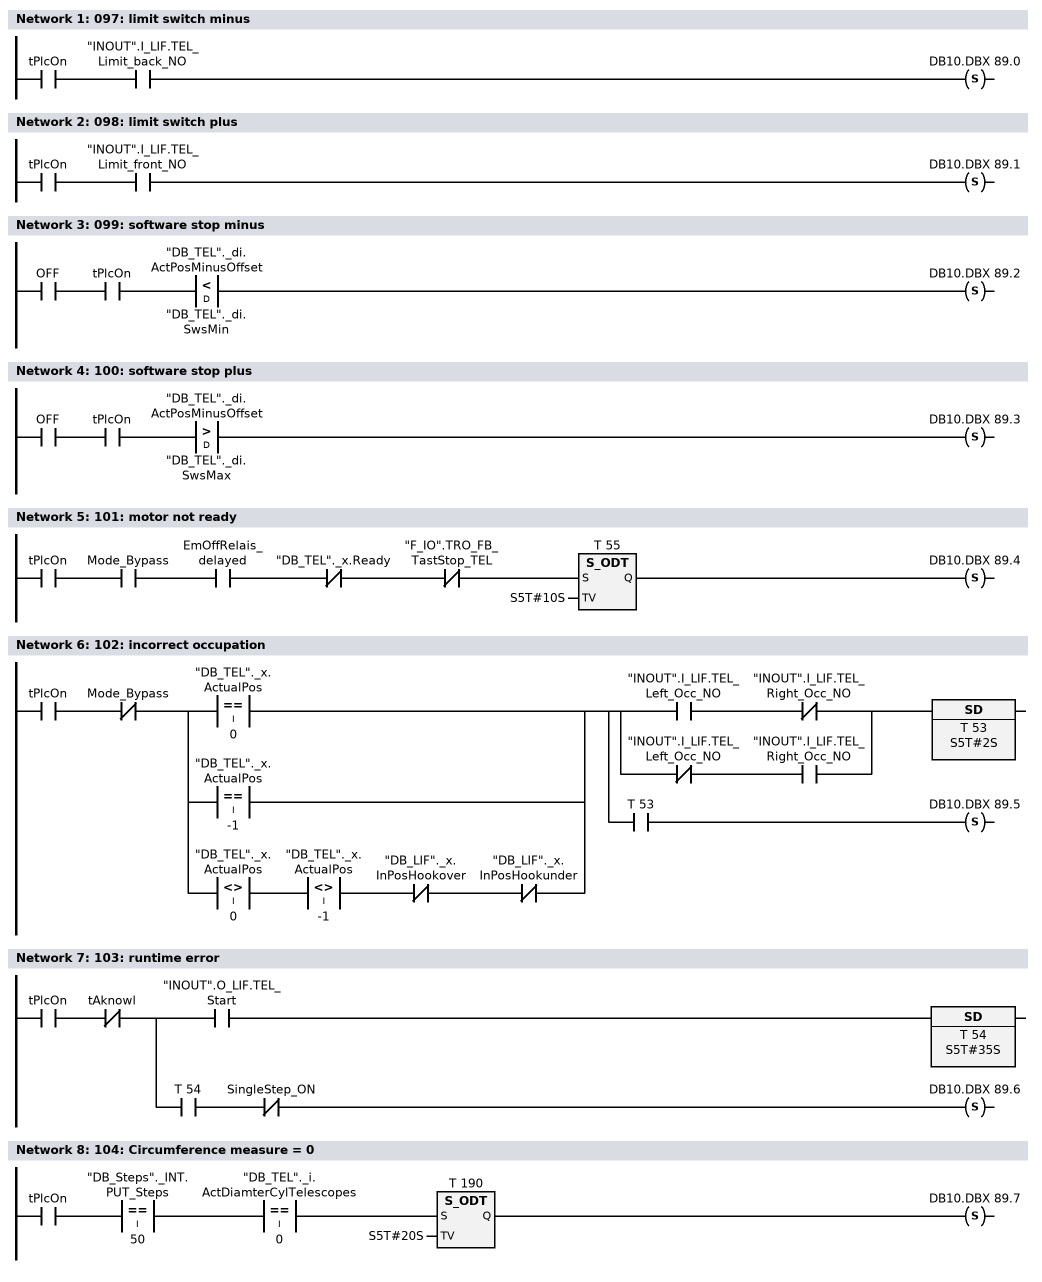
NETWORK
TITLE = 097: limit switch minus
      A     "tPlcOn";
      A     "INOUT".I_LIF.TEL_Limit_back_NO;
      S     DB10.DBX 89.0;
NETWORK
TITLE = 098: limit switch plus
      A     "tPlcOn";
      A     "INOUT".I_LIF.TEL_Limit_front_NO;
      S     DB10.DBX 89.1;
NETWORK
TITLE = 099: software stop minus
      A     "OFF";
      A     "tPlcOn";
      A(;
      L     "DB_TEL"._di.ActPosMinusOffset;
      L     "DB_TEL"._di.SwsMin;
      <D;
      );
      S     DB10.DBX 89.2;
NETWORK
TITLE = 100: software stop plus
      A     "OFF";
      A     "tPlcOn";
      A(;
      L     "DB_TEL"._di.ActPosMinusOffset;
      L     "DB_TEL"._di.SwsMax;
      >D;
      );
      S     DB10.DBX 89.3;
NETWORK
TITLE = 101: motor not ready
      A     "tPlcOn";
      A     "Mode_Bypass";
      A     "EmOffRelais_delayed";
      AN    "DB_TEL"._x.Ready;
      AN    "F_IO".TRO_FB_TastStop_TEL;
      L     S5T#10S;
      SD    T 55;
      NOP   0;
      NOP   0;
      NOP   0;
      A     T 55;
      S     DB10.DBX 89.4;
NETWORK
TITLE = 102: incorrect occupation
      A     "tPlcOn";
      AN    "Mode_Bypass";
      A(;
      O(;
      L     "DB_TEL"._x.ActualPos;
      L     0;
      ==I;
      );
      O(;
      L     "DB_TEL"._x.ActualPos;
      L     -1;
      ==I;
      );
      O;
      A(;
      L     "DB_TEL"._x.ActualPos;
      L     0;
      <>I;
      );
      A(;
      L     "DB_TEL"._x.ActualPos;
      L     -1;
      <>I;
      );
      AN    "DB_LIF"._x.InPosHookover;
      AN    "DB_LIF"._x.InPosHookunder;
      );
      =     L 0.0;
      A     L 0.0;
      A(;
      A     "INOUT".I_LIF.TEL_Left_Occ_NO;
      AN    "INOUT".I_LIF.TEL_Right_Occ_NO;
      O;
      AN    "INOUT".I_LIF.TEL_Left_Occ_NO;
      A     "INOUT".I_LIF.TEL_Right_Occ_NO;
      );
      L     S5T#2S;
      SD    T 53;
      A     L 0.0;
      A     T 53;
      S     DB10.DBX 89.5;
NETWORK
TITLE = 103: runtime error
      A     "tPlcOn";
      AN    "tAknowl";
      =     L 0.0;
      A     L 0.0;
      A     "INOUT".O_LIF.TEL_Start;
      L     S5T#35S;
      SD    T 54;
      A     L 0.0;
      A     T 54;
      AN    "SingleStep_ON";
      S     DB10.DBX 89.6;
NETWORK
TITLE = 104: Circumference measure = 0
      A     "tPlcOn";
      A(;
      L     "DB_Steps"._INT.PUT_Steps;
      L     50;
      ==I;
      );
      A(;
      L     "DB_TEL"._i.ActDiamterCylTelescopes;
      L     0;
      ==I;
      );
      L     S5T#20S;
      SD    T 190;
      NOP   0;
      NOP   0;
      NOP   0;
      A     T 190;
      S     DB10.DBX 89.7;
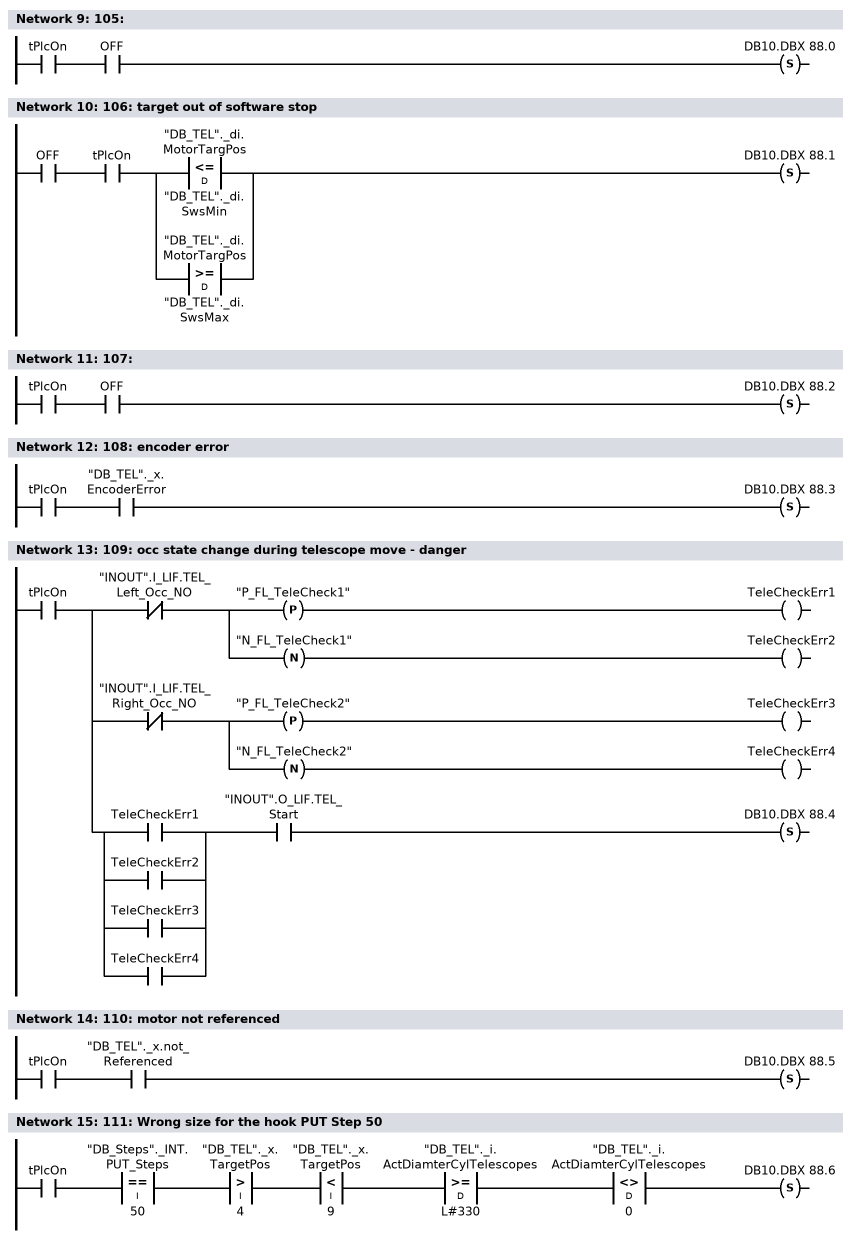
NETWORK
TITLE = 105:
      A     "tPlcOn";
      A     "OFF";
      S     DB10.DBX 88.0;
NETWORK
TITLE = 106: target out of software stop
      A     "OFF";
      A     "tPlcOn";
      A(;
      O(;
      L     "DB_TEL"._di.MotorTargPos;
      L     "DB_TEL"._di.SwsMin;
      <=D;
      );
      O(;
      L     "DB_TEL"._di.MotorTargPos;
      L     "DB_TEL"._di.SwsMax;
      >=D;
      );
      );
      S     DB10.DBX 88.1;
NETWORK
TITLE = 107: 
      A     "tPlcOn";
      A     "OFF";
      S     DB10.DBX 88.2;
NETWORK
TITLE = 108: encoder error
      A     "tPlcOn";
      A     "DB_TEL"._x.EncoderError;
      S     DB10.DBX 88.3;
NETWORK
TITLE = 109: occ state change during telescope move - danger
      A     "tPlcOn";
      =     L 0.0;
      A     L 0.0;
      AN    "INOUT".I_LIF.TEL_Left_Occ_NO;
      =     L 0.1;
      A     L 0.1;
      FP    "P_FL_TeleCheck1";
      =     "TeleCheckErr1";
      A     L 0.1;
      FN    "N_FL_TeleCheck1";
      =     "TeleCheckErr2";
      A     L 0.0;
      AN    "INOUT".I_LIF.TEL_Right_Occ_NO;
      =     L 0.1;
      A     L 0.1;
      FP    "P_FL_TeleCheck2";
      =     "TeleCheckErr3";
      A     L 0.1;
      FN    "N_FL_TeleCheck2";
      =     "TeleCheckErr4";
      A     L 0.0;
      A(;
      O     "TeleCheckErr1";
      O     "TeleCheckErr2";
      O     "TeleCheckErr3";
      O     "TeleCheckErr4";
      );
      A     "INOUT".O_LIF.TEL_Start;
      S     DB10.DBX 88.4;
NETWORK
TITLE = 110: motor not referenced
      A     "tPlcOn";
      A     "DB_TEL"._x.not_Referenced;
      S     DB10.DBX 88.5;
NETWORK
TITLE = 111: Wrong size for the hook PUT Step 50
//25.4 mm = 1 inch 
//
//40 inch = 1016
//34 inch = 863
//12 inch = 304
//10 inch = 254
      A     "tPlcOn";
      A(;
      L     "DB_Steps"._INT.PUT_Steps;
      L     50;
      ==I;
      );
      A(;
      L     "DB_TEL"._x.TargetPos;
      L     4;
      >I;
      );
      A(;
      L     "DB_TEL"._x.TargetPos;
      L     9;
      <I;
      );
      A(;
      L     "DB_TEL"._i.ActDiamterCylTelescopes;
      L     L#330;
      >=D;
      );
      A(;
      L     "DB_TEL"._i.ActDiamterCylTelescopes;
      L     0;
      <>D;
      );
      S     DB10.DBX 88.6;
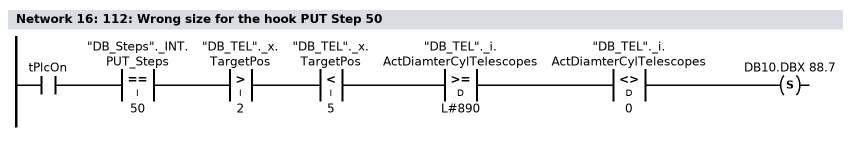
NETWORK
TITLE = 112: Wrong size for the hook PUT Step 50
      A     "tPlcOn";
      A(;
      L     "DB_Steps"._INT.PUT_Steps;
      L     50;
      ==I;
      );
      A(;
      L     "DB_TEL"._x.TargetPos;
      L     2;
      >I;
      );
      A(;
      L     "DB_TEL"._x.TargetPos;
      L     5;
      <I;
      );
      A(;
      L     "DB_TEL"._i.ActDiamterCylTelescopes;
      L     L#890;
      >=D;
      );
      A(;
      L     "DB_TEL"._i.ActDiamterCylTelescopes;
      L     0;
      <>D;
      );
      S     DB10.DBX 88.7;
END_FUNCTION

FUNCTION "Axis_TEL_Encoder" : VOID	// FC 240
TITLE = SSI Encoder Teleskope
//der SSI Drehgeber lässt sich nur auf 0 Preseten
//Faktor: 1mm = 7,31 Inkremente
//Mitte: damit es keine negativen Werte gibt, ist die Mittelstellung 2000mm
AUTHOR : bc
VERSION : 0.1
VAR_TEMP
  val : DINT ;
END_VAR
BEGIN
NETWORK
TITLE =
      L     "INOUT".I_LIF.TEL_Encoder;
      L     DW#16#0;	// offset
      +D;
      T     #val;
      L     DW#16#1FFFFFF;	// überlauf
      <=D;
      JC    m1;
      -D;
      T     #val;
m1:   L     #val;
      L     "DB_TEL"._di._FactorEncoder;
      /D;
      L     10;
      *D;
      T     "DB_TEL"._di._Enc_Korrektur;
      L     "DB_TEL"._di._PresetEncoder_mm;
      +D;
      T     "DB_TEL"._di._Enc_Korrektur;
      L     #val;
      L     L#10000000;
      >D;
      JC    gro0;
      JU    Korr;
gro0: L     "DB_TEL"._di._Enc_Korrektur;
      L     L#4596490;
      -D;
      T     "DB_TEL"._di._Enc_Korrektur;
Korr: NOP   0;
      L     "DB_TEL"._di._Enc_Korrektur;
      T     "DB_TEL"._di._ActEncoder_mm;
END_FUNCTION

FUNCTION "iPar_ServerCall" : VOID	// FC 900
TITLE = Trolley and Lift iParServer
VERSION : 0.1
VAR_TEMP
  tmp_date : DATE ;
  tmp_TOD : TIME_OF_DAY ;
  OB1_DATE_TIME : DATE_AND_TIME ;	//Date and time OB1 started
  on : BOOL ;
END_VAR
BEGIN
